// TIA Portal V20 export
// export: Created 2025-12-01T14:56:57.3436706Z, ExportSetting None, DisplayName Totally Integrated Automation Portal, DisplayVersion V20 Update 3, DisplayName TIA Portal Openness, DisplayVersion V20 Update 3, DisplayName TIA Portal Version Control Interface, DisplayVersion V20 Update 3, DisplayName STEP 7 Professional, DisplayVersion V20 Update 3, DisplayName STEP 7 Safety, DisplayVersion V20 Update 2, DisplayName WinCC Basic/Comfort/Advanced, DisplayVersion V20 Update 3, DisplayName WinCC Professional, DisplayVersion V20 Update 3, DisplayName WinCC Unified, DisplayVersion V20 Update 3
FUNCTION_BLOCK "FB376_DesPaletizador_Manual"   // FB376, LAD
TITLE = DesPaletizador Manual (Capas)
{ S7_Optimized_Access := 'FALSE' }
// stored: AutoNumber false, SetENOAutomatically false
   VAR_INPUT
      Maquina : UInt;   // Numero de Maquina
      ConfigDesPaletizador : "UDT_ConfigDesPaletizador";   // DB de Config de Velocidadad
      Robot_Habilitado : Bool;   // ROBOT >> Habilitado
      Robot_OutElevador : Bool;   // ROBOT >> Fuera de la Zona del Elevador
      Robot_PeticionSubir : Bool;   // ROBOT >> Peticion de Subir
      Robot_PeticionBajar : Bool;   // ROBOT >> Peticion de Bajar
      Robot_VelocidadElevador : Int;   // ROBOT >> Velocidad del Elevador
      ByteInicial : Int;   // Byte Inicial del Variador LENZE
      NodoNoPresente : Bool;   // Nodo No Presenye del Variador LENZE
      EnTension : Bool;   // Existe Tension en la Mesa
      Mantenimiento : Bool;   // Llave de Mantenimiento
      TermicoFreno : Bool;   // Termico del Freno
      Seg_UP : Bool;   // Seguridad Abajo de la Elevacion
      Seg_DOWN : Bool;   // Seguridad Abajo de la Elevacion
      pHsPisoCarga : Bool;   // Posicion del Piso de Carga
      pHsPisoDesCarga : Bool;   // Posicion del Piso de DesCarga
      Protrusion : Bool;   // pHs de Protrusion
      P_NuevaCapa : Bool;   // Peticion de Nueva Capa
      P_Subir : Bool;   // Pulsador de Subir
      P_Bajar : Bool;   // Pulsador de Bajar
      BarreraUp : Bool;   // Barrera del Nivel Superior
      pHsAnchura_01 : Bool;
      pHsAnchura_02 : Bool;
      pHsGalibo_01 : Bool;   // pHs de Control de Hueco Superior
      pHsGalibo_02 : Bool;   // pHs de Control de Hueco Superior
      pHsGalibo_03 : Bool;   // pHs de Control de Hueco Superior
      pHsGalibo_04 : Bool;   // pHs de Control de Hueco Superior
      pHsAlturaCota_01 : Bool;
      pHsAlturaCota_02 : Bool;
      pHsAlturaMax_01 : Bool;
      pHsAlturaMax_02 : Bool;
      RoturaCadena_01 : Bool;   // Rotura de Cadena
      RoturaCadena_02 : Bool;   // Rotura de Cadena
      RoturaCadena_03 : Bool;   // Rotura de Cadena
      RoturaCadena_04 : Bool;   // Rotura de Cadena
      FinDesPaletizado : Bool;   // Fin del Paletizado
      SubirManual : Bool;   // Subir en Manual
      BajarManual : Bool;   // Bajar en Manual
      Homming : Bool;
      EncoderIncremental : Bool;
      pHsReferenciaCero : Bool;   // phs de Referencia Cero
      V_TIM_Galibo : Time := T#1S;   // Morgan 14/02/19 500ms ->1s
      V_TIM_Protrusion : Int := 200;
      V_TOut_Elevacion : Int := 15000;
   END_VAR
   VAR_OUTPUT
      DesHabilitarBarreraUp : Bool;   // DesHabilitar Barrerra superior
      H_Puesto : Bool;   // Baliza de Paleta en Puesto
      DI3VarElev_pHsReferenciaCero : Bool;
   END_VAR
   VAR
      PosicionActual : Int;   // Posicion Actual
      PosicionDOWN : Int;   // Interna >> Posicion Abajo
      PosicionUP : Int;   // Interna >> Posicion Arriba
      PosicionOrden : Int;   // Orden >> Posicion A Ejecutar
      PosicionUltima : Int;   // Orden >> Ultima Posicion Enviada
      MemoPosicionActual : Int;   // Memoria >> Altura de la Carga
      MemoEventoDesPaletizado : Int;   // Memoria >> Evento Paletizado
      ConsignaFR : Int;   // Variador >> Consigna
      EstadoElevador : Word;   // Variador >> Estado
      Subject_Area : Word;   // Variador >> Subjet Area
      ID_Area : Word;   // Variador >> ID Area
      Orden : Bool;   // Orden >> Ejecutar
      FinOrden : Bool;   // Orden >> Fin Ejecucion
      PaletaEnPuesto : Bool;   // Interna >> Paleta En el Puesto
      MAQx_SinCapa : Bool;
      MemoCapaDinamico : Bool;
      FP_CapaDinamico : Bool;
      FN_CapaDinamico : Bool;
      InicioCapa : Int;
      FinalCapa : Int;
      MAQx_SinCota : Bool;
      MemoCotaDinamico : Bool;
      FP_CotaDinamico : Bool;
      MA_SubirPuesto : Bool;   // PUESTO >> Subir la Carga
      MA_BajarPuesto : Bool;   // PUESTO >> Bajar la Carga
      MA_Baliza : Bool;   // PUESTO >> Baliza
      PermisoMovElevador : Bool;   // Permiso Mover el Elevador
      PosCarga_OK : Bool;   // Posicionado en Carga
      PosDesCarga_OK : Bool;   // Posicionado en DesCargaCarga
      VarElev_MemoHomingAuto : Bool;   // Variador >>
      VarElev_ReferenciaOK : Bool;   // Variador >>
      VarElev_Error : Bool;   // Variador >>
      EventoInicioDesPaletizado : Bool;   // Evento >> Inicio DesPaletizado
      EventoFinalDesPaletizado : Bool;   // Evento >> Final DesPaletizado
      TIM_EsperaOrden { S7_SetPoint := 'True'} : TON_TIME;   // Orden >> TIM de Espera para Ejecutar
      TMPEnPisoCarga { S7_SetPoint := 'True'} : TON_TIME;
      TMPEnPisoDesCarga { S7_SetPoint := 'True'} : TON_TIME;
      TMP_EnTension { S7_SetPoint := 'True'} : "FB910_CNT_UHS";
      TOut_Elevacion { S7_SetPoint := 'True'} : "FB910_CNT_UHS";
      TIM_Protrusion { S7_SetPoint := 'True'} : "FB910_CNT_UHS";
      TIM_Galibo { S7_SetPoint := 'True'} : TON_TIME;
      TIM_EsperaErrorPosicion { S7_SetPoint := 'True'} : TON_TIME;
   END_VAR
   VAR_TEMP
      EstadoZonaMesa : "EstadoZona";
      EstadoZonaMaquina : "EstadoZona";
      EstadoVI : "EstadosMesa";
      EstadoMAQ : "EstadoMaquina_DesPaletizadoManual";
      DatosScada : "UDT_ScadaDatosMaquina";
      ConfigMAQ : "UDT_ConfigDesPaletizador";
      Auxiliares : Struct
         PosicionAbajo : Int;   // Posicion Abajo del Elevador
         AuxPosMax : Int;
         AuxPosMin : Int;
         Margen : Int;
         AuxAlturaMax : Int;
         AuxAlturaMin : Int;
      END_STRUCT;
      UT_Datos : Struct
         NumeroUT : UInt;
         CotaUT : Int;
         CapaUT : Int;
         SinUT : Bool;
         Con_DestinoUT : Bool;
         OK_DestinoUT : Bool;
      END_STRUCT;
      MovElevador : Struct
         NuevaPosicion : Int;
         AlturaVeloLentisima : Int;
         DestinoDOWN : Bool;   // Moviendose el elevador hacia la posicion de DOWN
         LentaDOWN : Bool;   // Activar velocidad lenta en el moviento hacia la posicion DOWN
         DestinoUP : Bool;   // Moviendose el elevador hacia la posicion de UP
         LentaUP : Bool;   // Activar velocidad lenta en el moviento hacia la posicion UP
         EnPisoAbajo : Bool;
         AlturaMax_OK : Bool;
         AlturaMin_OK : Bool;
      END_STRUCT;
      ZonaEnMarcha : Bool;
      ZonaEnReset : Bool;
      MAQ_Cargada : Bool;
      MAQ_Vacia : Bool;
      AlturaControlBarrerra : Int;
      AlturaCotaDefecto : Int;
      AlturaCapaDefecto : Int;
      AlturaCapaMinima : Int;
      AlturaCapaMaxima : Int;
      TempInt : Int;
   END_VAR
   VAR_TEMP   // added for the SCL form of the ladder/FBD networks
      _w1 : Bool;
      _w2 : Bool;
      _w3 : Bool;
   END_VAR
BEGIN

REGION Network 1: PARAMETROS ESPECIALES
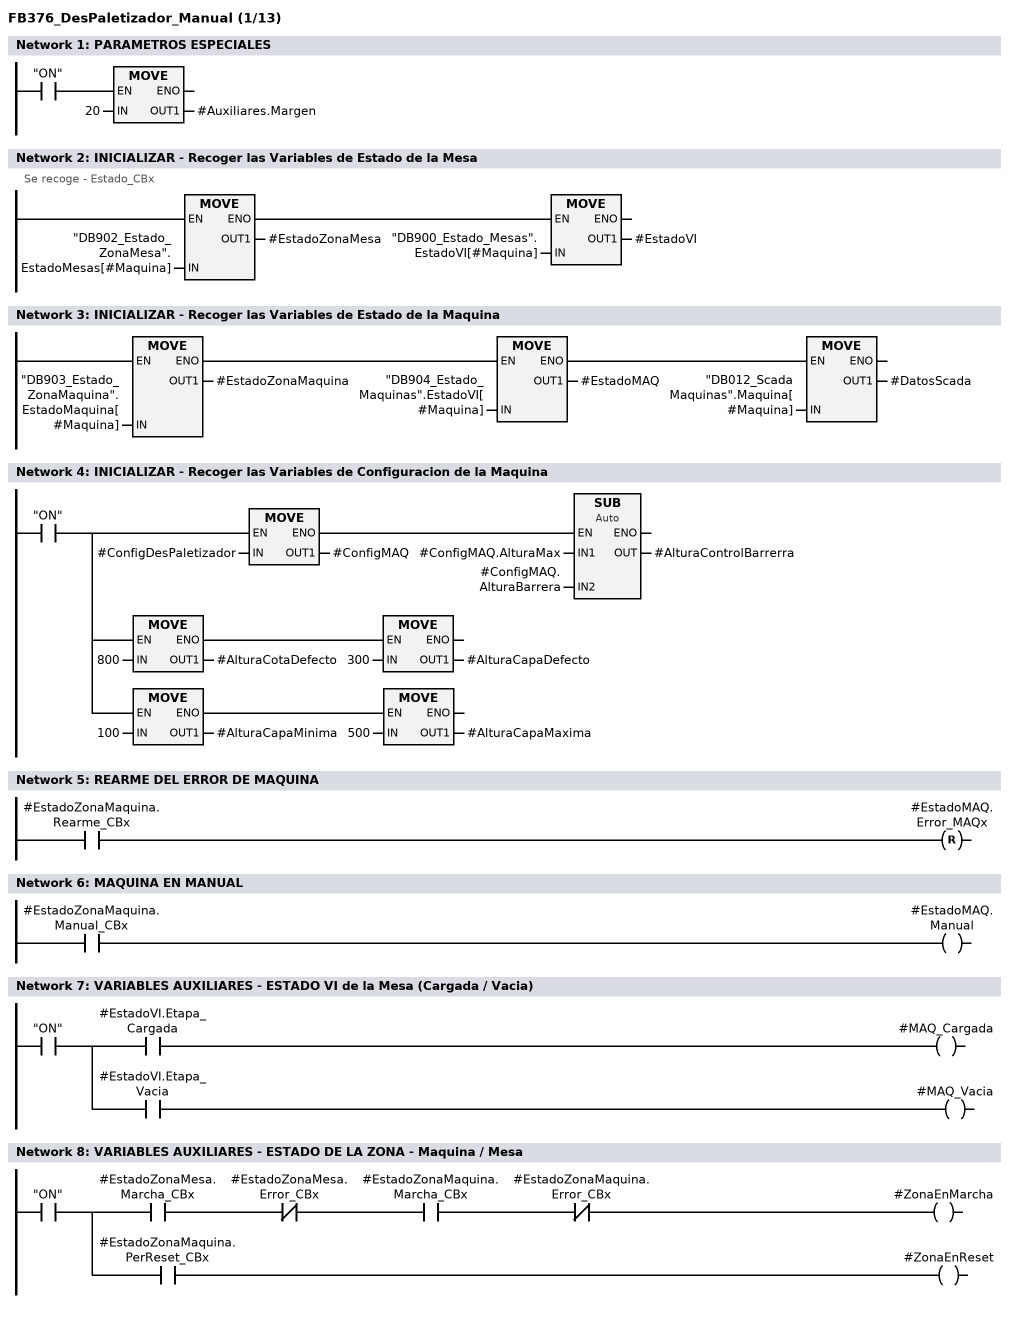
   RUNG wire#powerrail
      Contact( "ON" )
      { S7_GenerateENO := "TRUE" } Move(in := 20, out1 => #Auxiliares.Margen)
   END_RUNG
   // the same network as SCL:
   IF "ON" THEN #Auxiliares.Margen := 20; END_IF;
END_REGION

REGION Network 2: INICIALIZAR - Recoger las Variables de Estado de la Mesa
   // Se recoge - Estado_CBx
   RUNG wire#powerrail
      Move(in := "DB902_Estado_ZonaMesa".EstadoMesas[#Maquina], out1 => #EstadoZonaMesa)
      Move(in := "DB900_Estado_Mesas".EstadoVI[#Maquina], out1 => #EstadoVI)
   END_RUNG
   // the same network as SCL:
   #EstadoZonaMesa := "DB902_Estado_ZonaMesa".EstadoMesas[#Maquina];
   #EstadoVI := "DB900_Estado_Mesas".EstadoVI[#Maquina];
END_REGION

REGION Network 3: INICIALIZAR - Recoger las Variables de Estado de la Maquina
   RUNG wire#powerrail
      Move(in := "DB903_Estado_ZonaMaquina".EstadoMaquina[#Maquina], out1 => #EstadoZonaMaquina)
      Move(in := "DB904_Estado_Maquinas".EstadoVI[#Maquina], out1 => #EstadoMAQ)
      Move(in := "DB012_ScadaMaquinas".Maquina[#Maquina], out1 => #DatosScada)
   END_RUNG
   // the same network as SCL:
   #EstadoZonaMaquina := "DB903_Estado_ZonaMaquina".EstadoMaquina[#Maquina];
   #EstadoMAQ := "DB904_Estado_Maquinas".EstadoVI[#Maquina];
   #DatosScada := "DB012_ScadaMaquinas".Maquina[#Maquina];
END_REGION

REGION Network 4: INICIALIZAR - Recoger las Variables de Configuracion de la Maquina
   RUNG wire#powerrail
      Contact( "ON" )
      wire#w1
      Move(in := #ConfigDesPaletizador, out1 => #ConfigMAQ)
      Sub(in1 := #ConfigMAQ.AlturaMax, in2 := #ConfigMAQ.AlturaBarrera, out => #AlturaControlBarrerra)
   END_RUNG
   RUNG wire#w1
      Move(in := 800, out1 => #AlturaCotaDefecto)
      Move(in := 300, out1 => #AlturaCapaDefecto)
   END_RUNG
   RUNG wire#w1
      Move(in := 100, out1 => #AlturaCapaMinima)
      Move(in := 500, out1 => #AlturaCapaMaxima)
   END_RUNG
   // the same network as SCL:
   IF "ON" THEN
       #ConfigMAQ := #ConfigDesPaletizador;
       #AlturaControlBarrerra := #ConfigMAQ.AlturaMax - #ConfigMAQ.AlturaBarrera;
       #AlturaCotaDefecto := 800;
       #AlturaCapaDefecto := 300;
       #AlturaCapaMinima := 100;
       #AlturaCapaMaxima := 500;
   END_IF;
END_REGION

REGION Network 5: REARME DEL ERROR DE MAQUINA
   RUNG wire#powerrail
      Contact( #EstadoZonaMaquina.Rearme_CBx )
      R_Coil( #EstadoMAQ.Error_MAQx )
   END_RUNG
   // the same network as SCL:
   IF #EstadoZonaMaquina.Rearme_CBx THEN #EstadoMAQ.Error_MAQx := FALSE; END_IF;
END_REGION

REGION Network 6: MAQUINA EN MANUAL
   RUNG wire#powerrail
      Contact( #EstadoZonaMaquina.Manual_CBx )
      Coil( #EstadoMAQ.Manual )
   END_RUNG
   // the same network as SCL:
   #EstadoMAQ.Manual := #EstadoZonaMaquina.Manual_CBx;
END_REGION

REGION Network 7: VARIABLES AUXILIARES - ESTADO VI de la Mesa (Cargada / Vacia)
   RUNG wire#powerrail
      Contact( "ON" )
      wire#w1
      Contact( #EstadoVI.Etapa_Cargada )
      Coil( #MAQ_Cargada )
   END_RUNG
   RUNG wire#w1
      Contact( #EstadoVI.Etapa_Vacia )
      Coil( #MAQ_Vacia )
   END_RUNG
   // the same network as SCL:
   #MAQ_Cargada := "ON" AND #EstadoVI.Etapa_Cargada;
   #MAQ_Vacia := "ON" AND #EstadoVI.Etapa_Vacia;
END_REGION

REGION Network 8: VARIABLES AUXILIARES - ESTADO DE LA ZONA - Maquina / Mesa
   RUNG wire#powerrail
      Contact( "ON" )
      wire#w1
      Contact( #EstadoZonaMesa.Marcha_CBx )
      I_Contact( #EstadoZonaMesa.Error_CBx )
      Contact( #EstadoZonaMaquina.Marcha_CBx )
      I_Contact( #EstadoZonaMaquina.Error_CBx )
      Coil( #ZonaEnMarcha )
   END_RUNG
   RUNG wire#w1
      Contact( #EstadoZonaMaquina.PerReset_CBx )
      Coil( #ZonaEnReset )
   END_RUNG
   // the same network as SCL:
   #ZonaEnMarcha := "ON" AND #EstadoZonaMesa.Marcha_CBx AND NOT #EstadoZonaMesa.Error_CBx AND #EstadoZonaMaquina.Marcha_CBx AND NOT #EstadoZonaMaquina.Error_CBx;
   #ZonaEnReset := "ON" AND #EstadoZonaMaquina.PerReset_CBx;
END_REGION

NETWORK
TITLE = CONTROL DE RESET de Variables Auxiliares
/////////////////////////////////////////////////////////////////////////////
/////////////////////////////////////////////////////////////////////////////
// --- Si realiza un RESET hay que limpiar las variables

      SET;  // Reseteando la Maquina ?
      AN    #ZonaEnReset;
      JC    NoExiste_Reset;

      SET;
      R     #Orden;
      R     #PaletaEnPuesto;  // Variable del Puesto de Trabajo
      R     #MAQx_SinCota;
      R     #MAQx_SinCapa;

      L     0;
      T     #PosicionOrden;

NoExiste_Reset:NOP   0;



NETWORK
TITLE = CONTROL DE MOVIMIENTO DEL ELEVADOR - PROTOCOLO
/////////////////////////////////////////////////////////////////////////////
/////////////////////////////////////////////////////////////////////////////
// ---  Cierre del Protocolo

      SET;
      O     #Orden;  // - Hay que protocolo la Orden
      O     #FinOrden;  //   en ejecucion
      JCN   Final_ProtocoloOrden;
      SET;
      A     #Orden;  // - Hay que protocolo la Orden
      A     #FinOrden;  //   en ejecucion
      JCN   Final_ProtocoloOrden;

      L     0;  // -- Resetear Variables
      T     #PosicionOrden;

      SET;
      R     #Orden;

      JU    Final_ProtocoloOrden;


/////////////////////////////////////////////////////////////////////////////
/////////////////////////////////////////////////////////////////////////////
// ---  Final del Control

Final_ProtocoloOrden:NOP   0;


NETWORK
TITLE = RECOGER DATOS EXISTENTES DE LA UT
/////////////////////////////////////////////////////////////////////////////
/////////////////////////////////////////////////////////////////////////////
// ---  Datos de la UT en la Maquina
      L     0;
      T     #UT_Datos.CotaUT;
      T     #UT_Datos.CapaUT;

      SET;  // - Incializar datos de la UT
      R     #UT_Datos.OK_DestinoUT;
      R     #UT_Datos.Con_DestinoUT;
      S     #UT_Datos.SinUT;


/////////////////////////////////////////////////////////////////////////////
/////////////////////////////////////////////////////////////////////////////
// --- Comprobar si existen UT en la Mesa = Maquina

      L     "DB810_ColasMesas".Colas[#Maquina].UT_PrimeraMesa;
      T     #UT_Datos.NumeroUT;

      SET;  // No hay UT's ?
      L     #UT_Datos.NumeroUT;
      L     0;
      ==I;
      JC    Final_DatosUT;


/////////////////////////////////////////////////////////////////////////////
/////////////////////////////////////////////////////////////////////////////
// --- Recoger Datos
      SET;
      R     #UT_Datos.SinUT;  // --- Hay UT

      L     "DB815_UTs_Datos".UT[#UT_Datos.NumeroUT].CotaAltura;
      T     #UT_Datos.CotaUT;  // Altura de la Carga
      L     "DB815_UTs_Datos".UT[#UT_Datos.NumeroUT].Amarre;
      T     #UT_Datos.CapaUT;  // Capa

      SET;  // --- Comprobacion de Destino
      L     "DB812_UTs_Control".UT[#UT_Datos.NumeroUT].MesaDestino;
      L     0;
      ==I;
      JC    NoExiste_Destino;

      SET;  // --- Tiene Destino
      S     #UT_Datos.Con_DestinoUT;

      SET;  // --- Existe Destino de Evacuacion
      L     "DB812_UTs_Control".UT[#UT_Datos.NumeroUT].MesaDestino;
      L     "DB812_UTs_Control".UT[#UT_Datos.NumeroUT].MesaActual;
      <>I;
      S     #UT_Datos.OK_DestinoUT;

NoExiste_Destino:NOP   0;



/////////////////////////////////////////////////////////////////////////////
/////////////////////////////////////////////////////////////////////////////
// --- Control de la Altura de la UT

      L     #UT_Datos.CotaUT;  // - Control de la Cota
      L     0;
      <>I;
      JC    Existe_CotaUT;

      SET;
      S     #MAQx_SinCota;  // - Cota dianamica

      L     #AlturaCotaDefecto;  // - Valor de Defecto
      T     #UT_Datos.CotaUT;  // Se guarda ?
//      T     "DB815_DatosUT".Datos_UTs[#NumeroUT].CotaAltura

Existe_CotaUT:NOP   0;


/////////////////////////////////////////////////////////////////////////////
/////////////////////////////////////////////////////////////////////////////
// --- Control de la Capa de la UT

      L     #UT_Datos.CapaUT;  // - Control de la Capa
      L     0;
      <>I;
      JC    Existe_CapaUT;

      SET;
      S     #MAQx_SinCapa;  // - Capa dianamica

      L     #AlturaCapaDefecto;  //   Valor de Defecto
      T     #UT_Datos.CapaUT;  // Se guarda ?
      T     "DB815_UTs_Datos".UT[#UT_Datos.NumeroUT].Amarre;


Existe_CapaUT:NOP   0;
// - Altura para DesActivar el control de la Barrera
      L     #UT_Datos.CapaUT;
      L     200;
      +I;
      T     #AlturaControlBarrerra;


/////////////////////////////////////////////////////////////////////////////
/////////////////////////////////////////////////////////////////////////////
// --- Datos Recogidos
Final_DatosUT:NOP   0;  // --- Fin de los Datos de la UT

      SET;  // --- Configuracion del DesPaletizador
      AN    #UT_Datos.SinUT;  //     Dinamico
      JC    Existe_UT;

      R     #MAQx_SinCota;
      R     #MAQx_SinCapa;

Existe_UT:NOP   0;



REGION Network 12: VARIABLES AUXILIARES - Calculo de la Posicion Abajo del Elevador
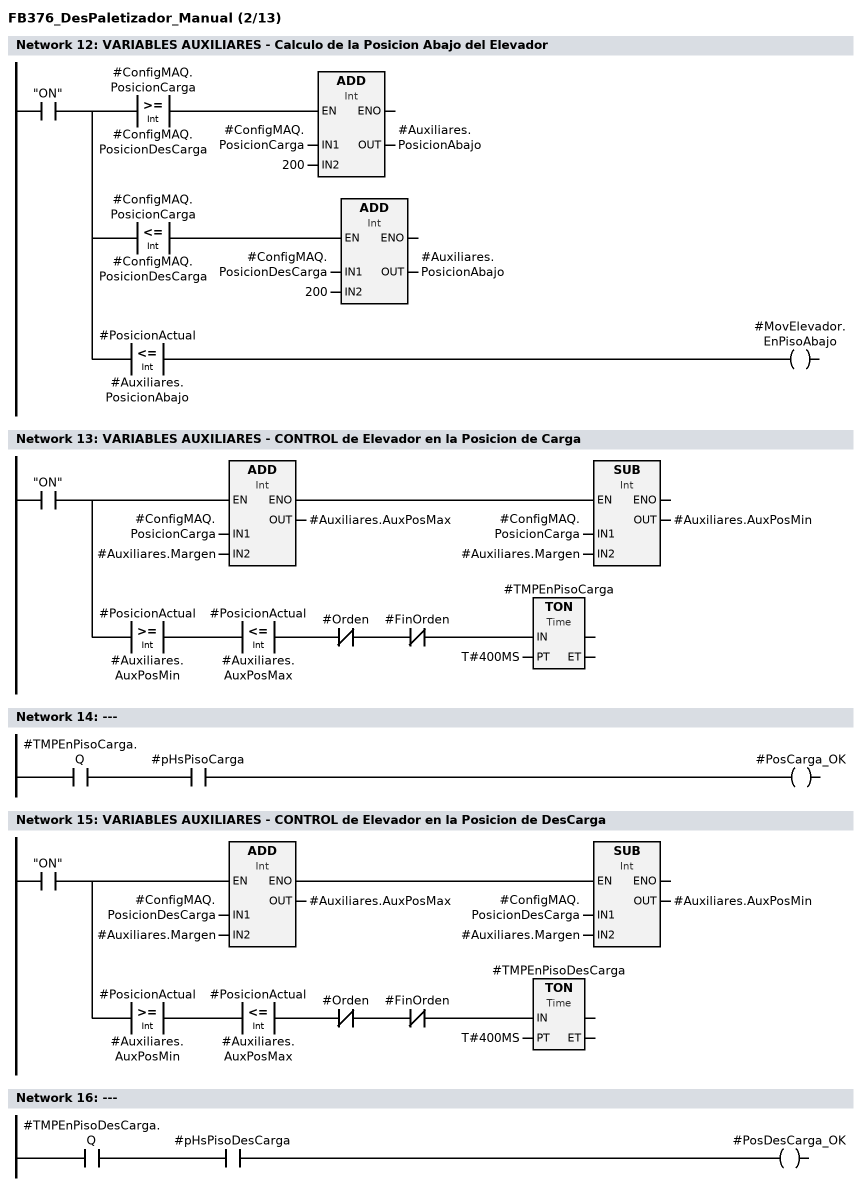
   RUNG wire#powerrail
      Contact( "ON" )
      wire#w1
      { S7_Templates := "SrcType := Int" } GE_Contact(in1 := #ConfigMAQ.PosicionCarga, in2 := #ConfigMAQ.PosicionDesCarga)
      { S7_Templates := "SrcType := Int"; S7_GenerateENO := "TRUE" } Add(in1 := #ConfigMAQ.PosicionCarga, in2 := 200, out => #Auxiliares.PosicionAbajo)
   END_RUNG
   RUNG wire#w1
      { S7_Templates := "SrcType := Int" } LE_Contact(in1 := #ConfigMAQ.PosicionCarga, in2 := #ConfigMAQ.PosicionDesCarga)
      { S7_Templates := "SrcType := Int"; S7_GenerateENO := "TRUE" } Add(in1 := #ConfigMAQ.PosicionDesCarga, in2 := 200, out => #Auxiliares.PosicionAbajo)
   END_RUNG
   RUNG wire#w1
      { S7_Templates := "SrcType := Int" } LE_Contact(in1 := #PosicionActual, in2 := #Auxiliares.PosicionAbajo)
      Coil( #MovElevador.EnPisoAbajo )
   END_RUNG
   // the same network as SCL:
   IF "ON" AND (#ConfigMAQ.PosicionCarga >= #ConfigMAQ.PosicionDesCarga) THEN
       #Auxiliares.PosicionAbajo := #ConfigMAQ.PosicionCarga + 200;
   END_IF;
   IF "ON" AND (#ConfigMAQ.PosicionCarga <= #ConfigMAQ.PosicionDesCarga) THEN
       #Auxiliares.PosicionAbajo := #ConfigMAQ.PosicionDesCarga + 200;
   END_IF;
   #MovElevador.EnPisoAbajo := "ON" AND (#PosicionActual <= #Auxiliares.PosicionAbajo);
END_REGION

REGION Network 13: VARIABLES AUXILIARES - CONTROL de Elevador en la Posicion de Carga
   RUNG wire#powerrail
      Contact( "ON" )
      wire#w1
      { S7_Templates := "SrcType := Int"; S7_GenerateENO := "TRUE" } Add(in1 := #ConfigMAQ.PosicionCarga, in2 := #Auxiliares.Margen, out => #Auxiliares.AuxPosMax)
      { S7_Templates := "SrcType := Int"; S7_GenerateENO := "TRUE" } Sub(in1 := #ConfigMAQ.PosicionCarga, in2 := #Auxiliares.Margen, out => #Auxiliares.AuxPosMin)
   END_RUNG
   RUNG wire#w1
      { S7_Templates := "SrcType := Int" } GE_Contact(in1 := #PosicionActual, in2 := #Auxiliares.AuxPosMin)
      { S7_Templates := "SrcType := Int" } LE_Contact(in1 := #PosicionActual, in2 := #Auxiliares.AuxPosMax)
      I_Contact( #Orden )
      I_Contact( #FinOrden )
      { S7_Templates := "time_type := Time" } #TMPEnPisoCarga.TON(pt := T#400MS, et =>)
   END_RUNG
   // the same network as SCL:
   // ENO of a box is taken as its EN; it also drops when the box reports an error
   IF "ON" THEN
       #Auxiliares.AuxPosMax := #ConfigMAQ.PosicionCarga + #Auxiliares.Margen;
       #Auxiliares.AuxPosMin := #ConfigMAQ.PosicionCarga - #Auxiliares.Margen;
   END_IF;
   #TMPEnPisoCarga(IN := "ON" AND (#PosicionActual >= #Auxiliares.AuxPosMin) AND (#PosicionActual <= #Auxiliares.AuxPosMax) AND NOT #Orden AND NOT #FinOrden,   // TON
                   PT := T#400MS);
END_REGION

REGION Network 14: ---
   RUNG wire#powerrail
      Contact( #TMPEnPisoCarga.Q )
      Contact( #pHsPisoCarga )
      Coil( #PosCarga_OK )
   END_RUNG
   // the same network as SCL:
   #PosCarga_OK := #TMPEnPisoCarga.Q AND #pHsPisoCarga;
END_REGION

REGION Network 15: VARIABLES AUXILIARES - CONTROL de Elevador en la Posicion de DesCarga
   RUNG wire#powerrail
      Contact( "ON" )
      wire#w1
      { S7_Templates := "SrcType := Int"; S7_GenerateENO := "TRUE" } Add(in1 := #ConfigMAQ.PosicionDesCarga, in2 := #Auxiliares.Margen, out => #Auxiliares.AuxPosMax)
      { S7_Templates := "SrcType := Int"; S7_GenerateENO := "TRUE" } Sub(in1 := #ConfigMAQ.PosicionDesCarga, in2 := #Auxiliares.Margen, out => #Auxiliares.AuxPosMin)
   END_RUNG
   RUNG wire#w1
      { S7_Templates := "SrcType := Int" } GE_Contact(in1 := #PosicionActual, in2 := #Auxiliares.AuxPosMin)
      { S7_Templates := "SrcType := Int" } LE_Contact(in1 := #PosicionActual, in2 := #Auxiliares.AuxPosMax)
      I_Contact( #Orden )
      I_Contact( #FinOrden )
      { S7_Templates := "time_type := Time" } #TMPEnPisoDesCarga.TON(pt := T#400MS, et =>)
   END_RUNG
   // the same network as SCL:
   // ENO of a box is taken as its EN; it also drops when the box reports an error
   IF "ON" THEN
       #Auxiliares.AuxPosMax := #ConfigMAQ.PosicionDesCarga + #Auxiliares.Margen;
       #Auxiliares.AuxPosMin := #ConfigMAQ.PosicionDesCarga - #Auxiliares.Margen;
   END_IF;
   #TMPEnPisoDesCarga(IN := "ON" AND (#PosicionActual >= #Auxiliares.AuxPosMin) AND (#PosicionActual <= #Auxiliares.AuxPosMax) AND NOT #Orden AND NOT #FinOrden,   // TON
                      PT := T#400MS);
END_REGION

REGION Network 16: ---
   RUNG wire#powerrail
      Contact( #TMPEnPisoDesCarga.Q )
      Contact( #pHsPisoDesCarga )
      Coil( #PosDesCarga_OK )
   END_RUNG
   // the same network as SCL:
   #PosDesCarga_OK := #TMPEnPisoDesCarga.Q AND #pHsPisoDesCarga;
END_REGION

REGION Network 17: VARIABLES AUXILIARES - CONTROL de Movimiento del Elevador en el Puesto de Trabajo (Maximo y Minimo)
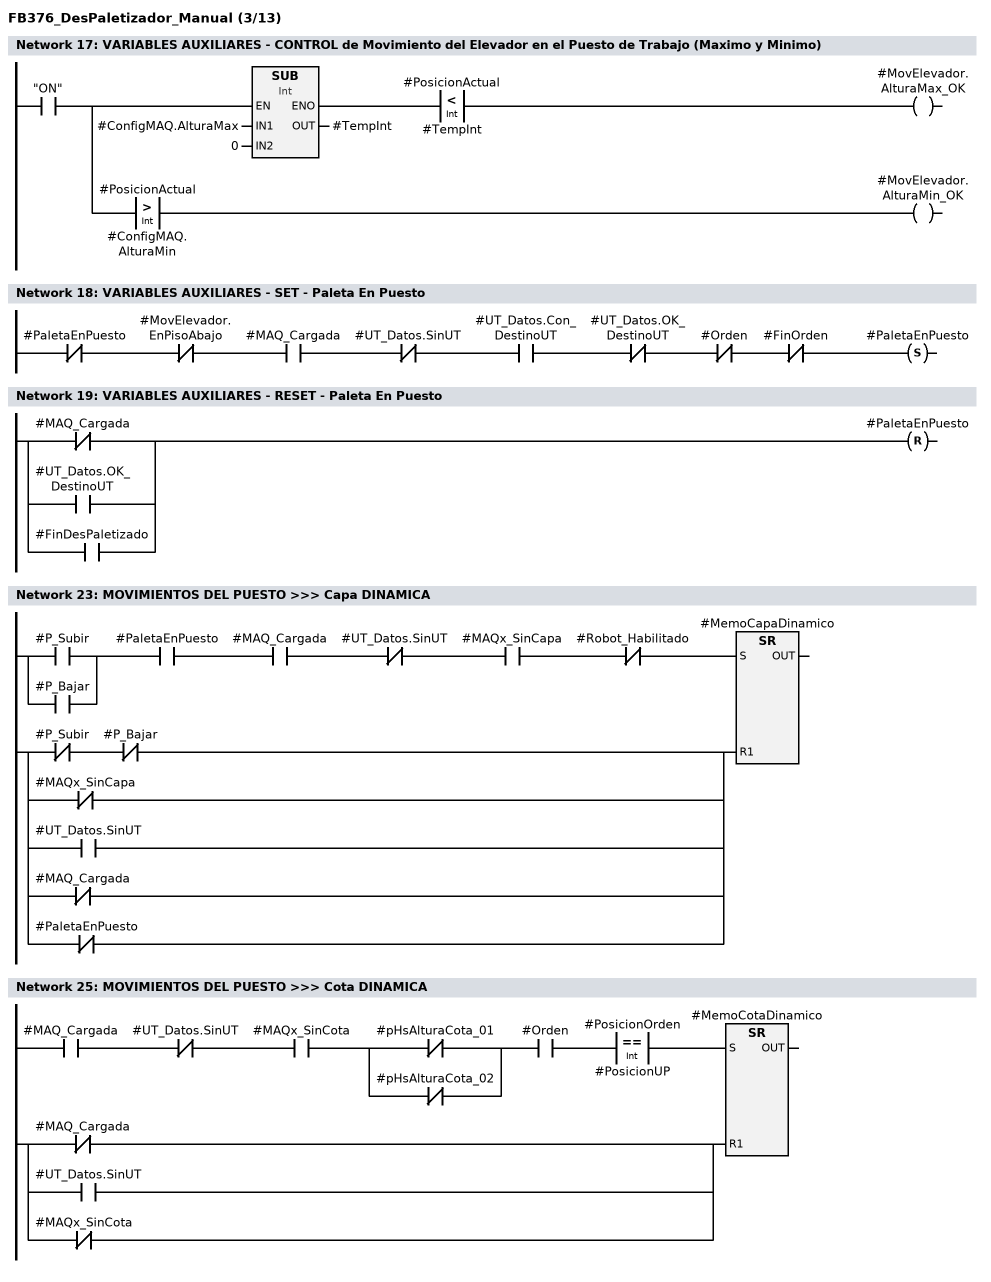
   RUNG wire#powerrail
      Contact( "ON" )
      wire#w1
      { S7_Templates := "SrcType := Int"; S7_GenerateENO := "TRUE" } Sub(in1 := #ConfigMAQ.AlturaMax, in2 := 0, out => #TempInt)
      { S7_Templates := "SrcType := Int" } LT_Contact(in1 := #PosicionActual, in2 := #TempInt)
      Coil( #MovElevador.AlturaMax_OK )
   END_RUNG
   RUNG wire#w1
      { S7_Templates := "SrcType := Int" } GT_Contact(in1 := #PosicionActual, in2 := #ConfigMAQ.AlturaMin)
      Coil( #MovElevador.AlturaMin_OK )
   END_RUNG
   // the same network as SCL:
   // ENO of a box is taken as its EN; it also drops when the box reports an error
   IF "ON" THEN #TempInt := #ConfigMAQ.AlturaMax - 0; END_IF;
   #MovElevador.AlturaMax_OK := "ON" AND (#PosicionActual < #TempInt);
   #MovElevador.AlturaMin_OK := "ON" AND (#PosicionActual > #ConfigMAQ.AlturaMin);
END_REGION

REGION Network 18: VARIABLES AUXILIARES - SET - Paleta En Puesto
   RUNG wire#powerrail
      I_Contact( #PaletaEnPuesto )
      I_Contact( #MovElevador.EnPisoAbajo )
      Contact( #MAQ_Cargada )
      I_Contact( #UT_Datos.SinUT )
      Contact( #UT_Datos.Con_DestinoUT )
      I_Contact( #UT_Datos.OK_DestinoUT )
      I_Contact( #Orden )
      I_Contact( #FinOrden )
      S_Coil( #PaletaEnPuesto )
   END_RUNG
   // the same network as SCL:
   IF NOT #PaletaEnPuesto AND NOT #MovElevador.EnPisoAbajo AND #MAQ_Cargada AND NOT #UT_Datos.SinUT AND #UT_Datos.Con_DestinoUT AND NOT #UT_Datos.OK_DestinoUT AND NOT #Orden AND NOT #FinOrden THEN
       #PaletaEnPuesto := TRUE;
   END_IF;
END_REGION

REGION Network 19: VARIABLES AUXILIARES - RESET - Paleta En Puesto
   RUNG wire#powerrail
      I_Contact( #MAQ_Cargada )
      wire#w1
      R_Coil( #PaletaEnPuesto )
   END_RUNG
   RUNG wire#powerrail
      Contact( #UT_Datos.OK_DestinoUT )
   END_RUNG wire#w1
   RUNG wire#powerrail
      Contact( #FinDesPaletizado )
   END_RUNG wire#w1
   // the same network as SCL:
   IF NOT #MAQ_Cargada OR #UT_Datos.OK_DestinoUT OR #FinDesPaletizado THEN #PaletaEnPuesto := FALSE; END_IF;
END_REGION

NETWORK
TITLE = MOVIMIENTOS DEL PUESTO >>> Control de Nueva CAPA
/////////////////////////////////////////////////////////////////////////////
/////////////////////////////////////////////////////////////////////////////
// ---  CONTROL DE NUEVA CAPA
      SET;
      A     #P_NuevaCapa;  // --- Se pulsado Nueva Capa ?
      A     #PaletaEnPuesto;  //     cuando esta la Paleta en el Puesto
      A     #MAQ_Cargada;  // --- Controles
      AN    #UT_Datos.SinUT;
      AN    #UT_Datos.OK_DestinoUT;
      AN    #FinDesPaletizado;
      AN    #Orden;
      AN    #FinOrden;
      AN    #Robot_Habilitado;
      JCN   Fin_ControlNuevaCapa;  // --- Realizar Nueva Capa ?


/////////////////////////////////////////////////////////////////////////////
/////////////////////////////////////////////////////////////////////////////
/////////////////////////////////////////////////////////////////////////////
      L     #PosicionActual;  // --- Calcular nueva posicion de parada
      L     #UT_Datos.CapaUT;  //     + Altura de Capa
      +D;
      T     #MovElevador.NuevaPosicion;

      L     #MovElevador.NuevaPosicion;  // --- Comprueba que no sobrepasa la altura maxima
      L     #ConfigMAQ.AlturaMax;
      <=I;
      JC    EjecutarOrden_NuevaCapa;

      L     #ConfigMAQ.AlturaMax;  // Lo maximo que se posiciona
      T     #MovElevador.NuevaPosicion;  // para trabajar

EjecutarOrden_NuevaCapa:NOP   0;
      L     #MovElevador.NuevaPosicion;
      T     #PosicionUP;  // - Guardar la Posicion UP
      T     #PosicionOrden;
      T     #PosicionUltima;

      S     #Orden;


/////////////////////////////////////////////////////////////////////////////
/////////////////////////////////////////////////////////////////////////////
/////////////////////////////////////////////////////////////////////////////
Fin_ControlNuevaCapa:NOP   0;



NETWORK
TITLE = CONTROL DE PULSADOR DE Subir >>> MA_SubirPuesto
/////////////////////////////////////////////////////////////////////////////
/////////////////////////////////////////////////////////////////////////////
// ---  Movimientos manuales desde el Puesto >>> SUBIR
      SET;
      A     #P_Subir;  // --- Orden de Subir el Elevador
      AN    #P_Bajar;
      AN    #P_NuevaCapa;
      A     #MovElevador.AlturaMax_OK;
      A     #PaletaEnPuesto;
      A     #MAQ_Cargada;  // --- Controles
      AN    #UT_Datos.SinUT;
      AN    #UT_Datos.OK_DestinoUT;
      AN    #FinDesPaletizado;
      AN    #Orden;
      AN    #FinOrden;
      AN    #Robot_Habilitado;
      =     #MA_SubirPuesto;




NETWORK
TITLE = CONTROL DE PULSADOR DE Bajar >>> MA_BajarPuesto
/////////////////////////////////////////////////////////////////////////////
/////////////////////////////////////////////////////////////////////////////
// ---  Movimientos manuales desde el Puesto >>> BAJAR
      SET;
      AN    #P_Subir;  // --- Orden de Bajar el Elevador
      A     #P_Bajar;
      AN    #P_NuevaCapa;
      A     #MovElevador.AlturaMin_OK;
      A     #PaletaEnPuesto;
      A     #MAQ_Cargada;  // --- Controles
      AN    #UT_Datos.SinUT;
      AN    #UT_Datos.OK_DestinoUT;
      AN    #FinDesPaletizado;
      AN    #Orden;
      AN    #FinOrden;
      AN    #Robot_Habilitado;
      =     #MA_BajarPuesto;



REGION Network 23: MOVIMIENTOS DEL PUESTO >>> Capa DINAMICA
   RUNG wire#powerrail
      Contact( #P_Subir )
      wire#w1
      Contact( #PaletaEnPuesto )
      Contact( #MAQ_Cargada )
      I_Contact( #UT_Datos.SinUT )
      Contact( #MAQx_SinCapa )
      I_Contact( #Robot_Habilitado )
      S_SR(operand := #MemoCapaDinamico, r1 := wire#w2)
   END_RUNG
   RUNG wire#powerrail
      Contact( #P_Bajar )
   END_RUNG wire#w1
   RUNG wire#powerrail
      I_Contact( #P_Subir )
      I_Contact( #P_Bajar )
   END_RUNG wire#w2
   RUNG wire#powerrail
      I_Contact( #MAQx_SinCapa )
   END_RUNG wire#w2
   RUNG wire#powerrail
      Contact( #UT_Datos.SinUT )
   END_RUNG wire#w2
   RUNG wire#powerrail
      I_Contact( #MAQ_Cargada )
   END_RUNG wire#w2
   RUNG wire#powerrail
      I_Contact( #PaletaEnPuesto )
   END_RUNG wire#w2
   // the same network as SCL:
   IF (#P_Subir OR #P_Bajar) AND #PaletaEnPuesto AND #MAQ_Cargada AND NOT #UT_Datos.SinUT AND #MAQx_SinCapa AND NOT #Robot_Habilitado THEN
       #MemoCapaDinamico := TRUE;   // SR flip-flop
   END_IF;
   IF (NOT #P_Subir AND NOT #P_Bajar) OR NOT #MAQx_SinCapa OR #UT_Datos.SinUT OR NOT #MAQ_Cargada OR NOT #PaletaEnPuesto THEN
       #MemoCapaDinamico := FALSE;
   END_IF;
END_REGION

NETWORK
TITLE = ---
/////////////////////////////////////////////////////////////////////////////
/////////////////////////////////////////////////////////////////////////////
/////////////////////////////////////////////////////////////////////////////
// --- Control Iniciales
      SET;  // --- Mirar Si existe control dianimico de CAPA
      AN    #MAQx_SinCapa;
      JC    Final_ControlCapaDinamica;
      SET;  // --- Existe UT
      A     #UT_Datos.SinUT;
      JC    Final_ControlCapaDinamica;


/////////////////////////////////////////////////////////////////////////////
/////////////////////////////////////////////////////////////////////////////
/////////////////////////////////////////////////////////////////////////////
// --- Control del Calculo de Capa Dinamica
      SET;
      A     #MemoCapaDinamico;
      FP    #FP_CapaDinamico;  // --- FP del Calculo de Capa
      JC    Inicio_CalculoCapaDianamica;

      SET;
      A     #MemoCapaDinamico;
      FN    #FN_CapaDinamico;  // --- FP del Calculo de Capa
      JC    Final_CalculoCapaDianamica;

      JU    Final_ControlCapaDinamica;


/////////////////////////////////////////////////////////////////////////////
/////////////////////////////////////////////////////////////////////////////
/////////////////////////////////////////////////////////////////////////////
//--- Inicio del Calculo de Capa
Inicio_CalculoCapaDianamica:NOP   0;
      L     #PosicionActual;
      T     #InicioCapa;
      JU    Final_ControlCapaDinamica;


/////////////////////////////////////////////////////////////////////////////
/////////////////////////////////////////////////////////////////////////////
/////////////////////////////////////////////////////////////////////////////
//--- Fin del Calculo de Capa
Final_CalculoCapaDianamica:NOP   0;
      L     #PosicionActual;
      T     #FinalCapa;

      L     #FinalCapa;  // --- Altura de nueva capa
      L     #InicioCapa;
      -I;
      L     #UT_Datos.CapaUT;
      +I;
      T     #UT_Datos.CapaUT;

/////////////////////////////////////////////////////////////////////////////
//--- Altura Minima de Capa ? (Altura Capa Minima)
      L     #UT_Datos.CapaUT;
      L     #AlturaCapaMinima;
      >=I;
      JC    MimimoOK_ControlCapaDinamica;

      L     #AlturaCapaMinima;
      T     #UT_Datos.CapaUT;
MimimoOK_ControlCapaDinamica:NOP   0;

/////////////////////////////////////////////////////////////////////////////
//--- Altura Maxima de Capa ? (Altura Capa Maxima)
      L     #UT_Datos.CapaUT;  // --- Altura MAxima de Capa
      L     #AlturaCapaMaxima;  //     Max.Capa por defecto
      <=I;
      JC    MaximoOK_ControlCapaDinamica;

      L     #AlturaCapaMaxima;
      T     #UT_Datos.CapaUT;
MaximoOK_ControlCapaDinamica:NOP   0;

//--- Guardar la Nueva Capa de la UT
      L     #UT_Datos.CapaUT;
      T     "DB815_UTs_Datos".UT[#UT_Datos.NumeroUT].Amarre;


/////////////////////////////////////////////////////////////////////////////
/////////////////////////////////////////////////////////////////////////////
/////////////////////////////////////////////////////////////////////////////
Final_ControlCapaDinamica:NOP   0;



REGION Network 25: MOVIMIENTOS DEL PUESTO >>> Cota DINAMICA
   RUNG wire#powerrail
      Contact( #MAQ_Cargada )
      I_Contact( #UT_Datos.SinUT )
      Contact( #MAQx_SinCota )
      wire#w1
      I_Contact( #pHsAlturaCota_01 )
      wire#w2
      Contact( #Orden )
      { S7_Templates := "SrcType := Int" } EQ_Contact(in1 := #PosicionOrden, in2 := #PosicionUP)
      S_SR(operand := #MemoCotaDinamico, r1 := wire#w3)
   END_RUNG
   RUNG wire#w1
      I_Contact( #pHsAlturaCota_02 )
   END_RUNG wire#w2
   RUNG wire#powerrail
      I_Contact( #MAQ_Cargada )
   END_RUNG wire#w3
   RUNG wire#powerrail
      Contact( #UT_Datos.SinUT )
   END_RUNG wire#w3
   RUNG wire#powerrail
      I_Contact( #MAQx_SinCota )
   END_RUNG wire#w3
   // the same network as SCL:
   IF #MAQ_Cargada AND NOT #UT_Datos.SinUT AND #MAQx_SinCota AND (NOT #pHsAlturaCota_01 OR NOT #pHsAlturaCota_02) AND #Orden AND (#PosicionOrden = #PosicionUP) THEN
       #MemoCotaDinamico := TRUE;   // SR flip-flop
   END_IF;
   IF NOT #MAQ_Cargada OR #UT_Datos.SinUT OR NOT #MAQx_SinCota THEN #MemoCotaDinamico := FALSE; END_IF;
END_REGION

NETWORK
TITLE = ---
/////////////////////////////////////////////////////////////////////////////
/////////////////////////////////////////////////////////////////////////////
/////////////////////////////////////////////////////////////////////////////
// --- Control Iniciales
      SET;  // --- Mirar Si existe control dianimico de Cota
      AN    #MAQx_SinCota;
      JC    Final_ControlCotaDinamica;
      SET;  // --- Existe UT
      A     #UT_Datos.SinUT;
      JC    Final_ControlCotaDinamica;


/////////////////////////////////////////////////////////////////////////////
/////////////////////////////////////////////////////////////////////////////
/////////////////////////////////////////////////////////////////////////////
// --- Control de Altura de la Paleta COTA--> Solo la primera vez
      SET;
      A     #MemoCotaDinamico;
      FP    #FP_CotaDinamico;  // --- FP del Calculo de Cota
      JCN   Final_ControlCotaDinamica;

/////////////////////////////////////////////////////////////////////////////
// --- Nueva Posicion de Parada
      L     #ConfigMAQ.AlturaMax;
      L     #ConfigMAQ.AlturaGalibo;
      -I;
      L     #PosicionActual;
      +I;
      L     #UT_Datos.CapaUT;
      +I;
//     L     #AlturaPaleta        // --- NO NECESARIO ???
//      +I
      T     #MovElevador.NuevaPosicion;

/////////////////////////////////////////////////////////////////////////////
//--- Altura Maxima de Cota ? (Altura Maxima)
      L     #MovElevador.NuevaPosicion;  // --- Comprueba que no sobrepasa
      L     #ConfigMAQ.AlturaMax;  //     la altura maxima
      <=I;
      JC    MaximoOK_ControlCotaDinamica;

      L     #ConfigMAQ.AlturaMax;  // Lo maximo que se posiciona
      T     #MovElevador.NuevaPosicion;  // para trabajar

MaximoOK_ControlCotaDinamica:NOP   0;
      L     #MovElevador.NuevaPosicion;
      T     #PosicionOrden;
      T     #PosicionUltima;
      T     #PosicionUP;


/////////////////////////////////////////////////////////////////////////////
/////////////////////////////////////////////////////////////////////////////
/////////////////////////////////////////////////////////////////////////////
Final_ControlCotaDinamica:NOP   0;



NETWORK
TITLE = GESTION DE ORDENES DE POSICIONADO >>> POSICIONAR el Elevador --- Controles Iniciales
/////////////////////////////////////////////////////////////////////////////
/////////////////////////////////////////////////////////////////////////////
// --- Controles iniciales
      SET;  // Ya esta la Paleta en el Puesto ?
      A     #PaletaEnPuesto;
      JC    Final_ControlOrdenes;

      SET;  // Esta en Marcha ?
      AN    #ZonaEnMarcha;
      JC    Final_ControlOrdenes;

      SET;  // Hay Orden en Curso ?
      A     #Orden;
      O     #FinOrden;
      JC    Final_ControlOrdenes;




NETWORK
TITLE = ---- Distribucion para Ordenes de Posicionado
/////////////////////////////////////////////////////////////////////////////
/////////////////////////////////////////////////////////////////////////////
/////////////////////////////////////////////////////////////////////////////
/////////////////////////////////////////////////////////////////////////////
// --- CONTROL DE ORDENES >>> La Paleta No esta en el Puesto


// --- Posicionar para CARGAR
      SET;
      A     #MAQ_Vacia;  // Esta VACIA
      A     #UT_Datos.SinUT;  // No hay UT
      AN    #MovElevador.EnPisoAbajo;
      JC    Posicionar_CARGA;


// --- Posicionar en el PUESTO DE TRABAJO
      SET;
      A     #MAQ_Cargada;  // Esta CARGADA
      AN    #FinDesPaletizado;  // Sin ORDEN
      AN    #UT_Datos.SinUT;  // Hay UT
      AN    #UT_Datos.OK_DestinoUT;  // No tiene DESTINO
      A     #UT_Datos.Con_DestinoUT;
      A     #MovElevador.EnPisoAbajo;
      AN    #Robot_Habilitado;
      JC    Posicionar_ARRIBA_SIN_ROBOT;

      SET;
      A     #MAQ_Cargada;  // Esta CARGADA
      AN    #FinDesPaletizado;  // Sin ORDEN
      AN    #UT_Datos.SinUT;  // Hay UT
      AN    #UT_Datos.OK_DestinoUT;  // No tiene DESTINO
      A     #UT_Datos.Con_DestinoUT;
      A     #MovElevador.EnPisoAbajo;
      A     #Robot_Habilitado;
      JC    Posicionar_ARRIBA_CON_ROBOT;


// --- Posicionar para DESCARGAR
      SET;
      A     #MAQ_Cargada;  // Esta CARGADA
      A     #FinDesPaletizado;  // Con ORDEN
      AN    #UT_Datos.SinUT;  // Hay UT
      AN    #MovElevador.EnPisoAbajo;
      JC    Posicionar_DESCARGA;

      SET;
      A     #MAQ_Cargada;  // Esta CARGADA
      AN    #FinDesPaletizado;  // Sin ORDEN
      AN    #UT_Datos.SinUT;  // Hay UT
      A     #UT_Datos.OK_DestinoUT;  // Tiene DESTINO
      A     #UT_Datos.Con_DestinoUT;
      AN    #MovElevador.EnPisoAbajo;
      JC    Posicionar_DESCARGA;

      JU    Final_ControlOrdenes;  // No hay Ordenes



NETWORK
TITLE = ---- Ejecutar Ordenes de Posicionado
/////////////////////////////////////////////////////////////////////////////
/////////////////////////////////////////////////////////////////////////////
/////////////////////////////////////////////////////////////////////////////
/////////////////////////////////////////////////////////////////////////////
// ---  POSICIONAR PARA LA CARGA
Posicionar_CARGA:NOP   0;
      SET;
      S     #Orden;

      L     #ConfigMAQ.PosicionCarga;  // --- Enviar orden de Reposo
      T     #PosicionDOWN;  //     Piso de ABAJO
      T     #PosicionOrden;
      T     #PosicionUltima;

      JU    Final_ControlOrdenes;


/////////////////////////////////////////////////////////////////////////////
/////////////////////////////////////////////////////////////////////////////
/////////////////////////////////////////////////////////////////////////////
/////////////////////////////////////////////////////////////////////////////
// ---  POSICIONAR PARA LA DESCARGA
Posicionar_DESCARGA:NOP   0;
      SET;
      S     #Orden;

      L     #ConfigMAQ.PosicionDesCarga;  // --- Enviar orden de Reposo
      T     #PosicionDOWN;  //     Piso de ABAJO
      T     #PosicionOrden;
      T     #PosicionUltima;

      JU    Final_ControlOrdenes;


/////////////////////////////////////////////////////////////////////////////
/////////////////////////////////////////////////////////////////////////////
/////////////////////////////////////////////////////////////////////////////
/////////////////////////////////////////////////////////////////////////////
// ---  POSICIONAR EN EL PUESTO DE TRABAJO >>> SIN ROBOT
Posicionar_ARRIBA_SIN_ROBOT:NOP   0;
      SET;
      S     #Orden;

      L     #ConfigMAQ.AlturaMax;  // --- Altura Inicial en el Puesto de Trabajo
      L     #UT_Datos.CotaUT;  //     Altura a posicionarse =
      -I;  // = AlturaMaxima - Cota
      L     #UT_Datos.CapaUT;  // + Capa
      +I;
      L     #ConfigMAQ.AlturaPaleta;  // + Altura de Paleta
      +I;
      T     #MovElevador.NuevaPosicion;

//--- Altura Maxima ?
      L     #MovElevador.NuevaPosicion;  // --- Comprueba que no sobrepasa
      L     #ConfigMAQ.AlturaMax;  //     la altura maxima
      <=I;
      JC    MaximoOK_Posicionar_ARRIBA_SIN_ROBOT;

      L     #ConfigMAQ.AlturaMax;  // Lo maximo que se posiciona
      T     #MovElevador.NuevaPosicion;  // para trabajar

MaximoOK_Posicionar_ARRIBA_SIN_ROBOT:NOP   0;
      L     #MovElevador.NuevaPosicion;
      T     #PosicionUP;
      T     #PosicionOrden;
      T     #PosicionUltima;

      JU    Final_ControlOrdenes;
/////////////////////////////////////////////////////////////////////////////
/////////////////////////////////////////////////////////////////////////////
/////////////////////////////////////////////////////////////////////////////
/////////////////////////////////////////////////////////////////////////////
// ---  POSICIONAR EN EL PUESTO DE TRABAJO >>> SIN ROBOT
Posicionar_ARRIBA_CON_ROBOT:NOP   0;
      SET;
      S     #Orden;

      L     #ConfigMAQ.AlturaMax;  // --- Altura Inicial en el Puesto de Trabajo
      L     #UT_Datos.CotaUT;  //     Altura a posicionarse =
      -I;  // = AlturaMaxima - Cota
//      L     #UT_Datos.CapaUT     // + Capa
//      +I
      L     #ConfigMAQ.AlturaPaleta;  // + Altura de Paleta
      +I;
      T     #MovElevador.NuevaPosicion;

//--- Altura Maxima ?
      L     #MovElevador.NuevaPosicion;  // --- Comprueba que no sobrepasa
      L     #ConfigMAQ.AlturaMax;  //     la altura maxima
      <=I;
      JC    MaximoOK_Posicionar_ARRIBA_CON_ROBOT;

      L     #ConfigMAQ.AlturaMax;  // Lo maximo que se posiciona
      T     #MovElevador.NuevaPosicion;  // para trabajar

MaximoOK_Posicionar_ARRIBA_CON_ROBOT:NOP   0;
      L     #MovElevador.NuevaPosicion;
      T     #PosicionUP;
      T     #PosicionOrden;
      T     #PosicionUltima;

      JU    Final_ControlOrdenes;



NETWORK
TITLE = ---- Final
/////////////////////////////////////////////////////////////////////////////
/////////////////////////////////////////////////////////////////////////////
/////////////////////////////////////////////////////////////////////////////
/////////////////////////////////////////////////////////////////////////////
// --- Final del Control de Ordenes
Final_ControlOrdenes:NOP   0;



REGION Network 31: CONTROL DE FRENCUENCIA DE POSICIONADO DEL VATIADOR DEL ELEVADOR
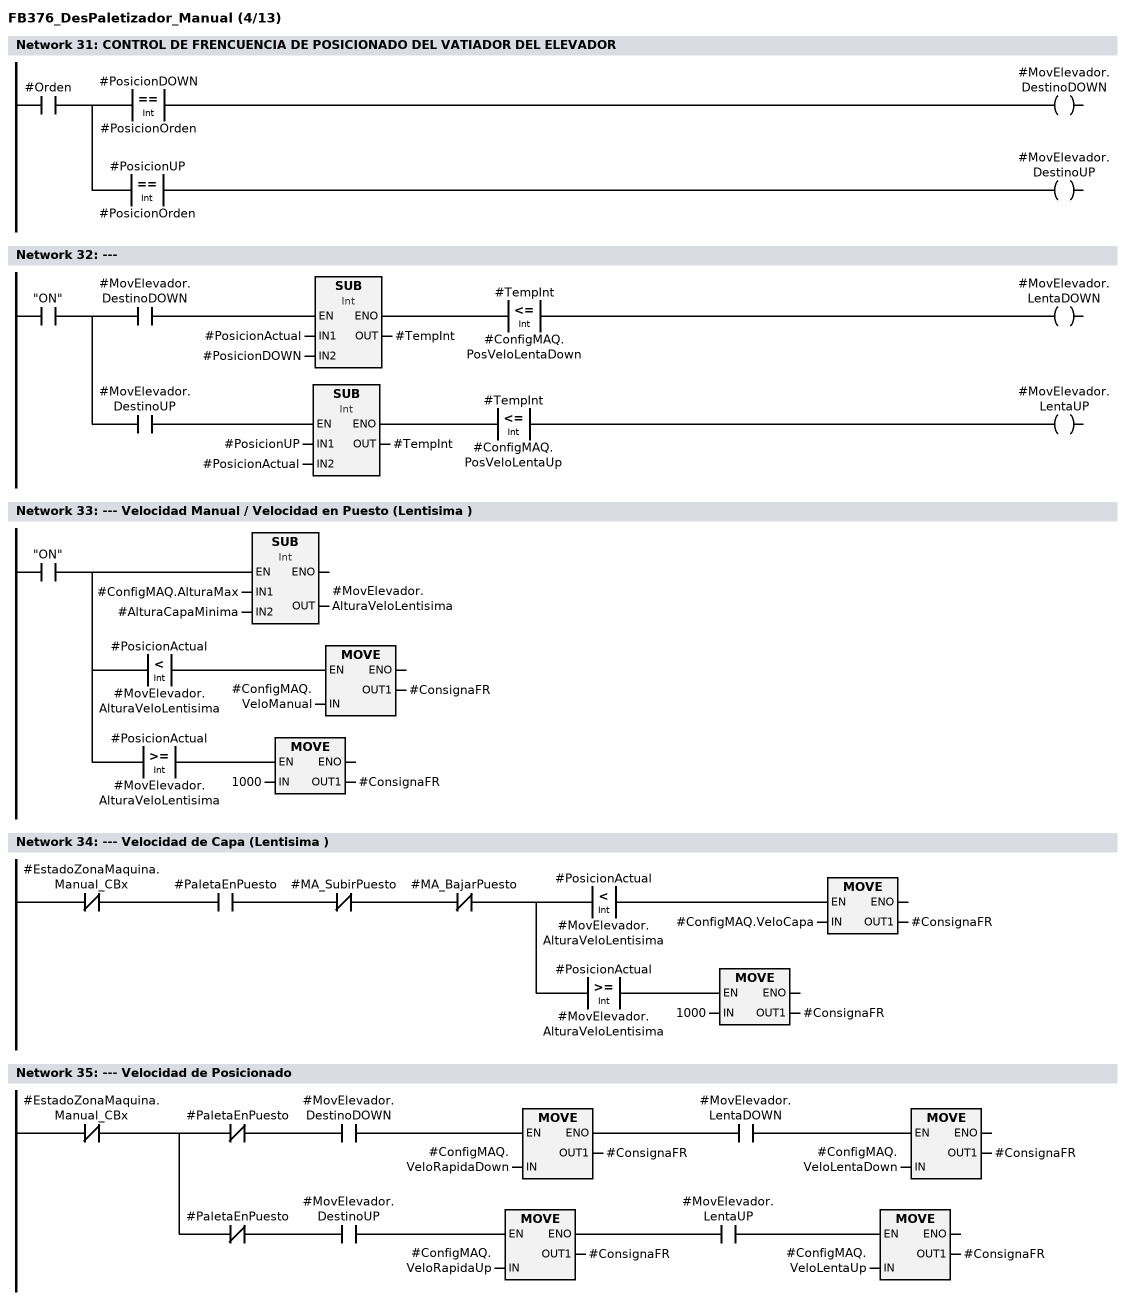
   RUNG wire#powerrail
      Contact( #Orden )
      wire#w1
      { S7_Templates := "SrcType := Int" } EQ_Contact(in1 := #PosicionDOWN, in2 := #PosicionOrden)
      Coil( #MovElevador.DestinoDOWN )
   END_RUNG
   RUNG wire#w1
      { S7_Templates := "SrcType := Int" } EQ_Contact(in1 := #PosicionUP, in2 := #PosicionOrden)
      Coil( #MovElevador.DestinoUP )
   END_RUNG
   // the same network as SCL:
   #MovElevador.DestinoDOWN := #Orden AND (#PosicionDOWN = #PosicionOrden);
   #MovElevador.DestinoUP := #Orden AND (#PosicionUP = #PosicionOrden);
END_REGION

REGION Network 32: ---
   RUNG wire#powerrail
      Contact( "ON" )
      wire#w1
      Contact( #MovElevador.DestinoDOWN )
      { S7_Templates := "SrcType := Int"; S7_GenerateENO := "TRUE" } Sub(in1 := #PosicionActual, in2 := #PosicionDOWN, out => #TempInt)
      { S7_Templates := "SrcType := Int" } LE_Contact(in1 := #TempInt, in2 := #ConfigMAQ.PosVeloLentaDown)
      Coil( #MovElevador.LentaDOWN )
   END_RUNG
   RUNG wire#w1
      Contact( #MovElevador.DestinoUP )
      { S7_Templates := "SrcType := Int"; S7_GenerateENO := "TRUE" } Sub(in1 := #PosicionUP, in2 := #PosicionActual, out => #TempInt)
      { S7_Templates := "SrcType := Int" } LE_Contact(in1 := #TempInt, in2 := #ConfigMAQ.PosVeloLentaUp)
      Coil( #MovElevador.LentaUP )
   END_RUNG
   // the same network as SCL:
   // ENO of a box is taken as its EN; it also drops when the box reports an error
   #_w1 := "ON" AND #MovElevador.DestinoDOWN;
   IF #_w1 THEN #TempInt := #PosicionActual - #PosicionDOWN; END_IF;
   #MovElevador.LentaDOWN := #_w1 AND (#TempInt <= #ConfigMAQ.PosVeloLentaDown);
   #_w2 := "ON" AND #MovElevador.DestinoUP;
   IF #_w2 THEN #TempInt := #PosicionUP - #PosicionActual; END_IF;
   #MovElevador.LentaUP := #_w2 AND (#TempInt <= #ConfigMAQ.PosVeloLentaUp);
END_REGION

REGION Network 33: --- Velocidad Manual / Velocidad en Puesto (Lentisima )
   RUNG wire#powerrail
      Contact( "ON" )
      wire#w1
      { S7_Templates := "SrcType := Int"; S7_GenerateENO := "TRUE" } Sub(in1 := #ConfigMAQ.AlturaMax, in2 := #AlturaCapaMinima, out => #MovElevador.AlturaVeloLentisima)
   END_RUNG
   RUNG wire#w1
      { S7_Templates := "SrcType := Int" } LT_Contact(in1 := #PosicionActual, in2 := #MovElevador.AlturaVeloLentisima)
      { S7_GenerateENO := "TRUE" } Move(in := #ConfigMAQ.VeloManual, out1 => #ConsignaFR)
   END_RUNG
   RUNG wire#w1
      { S7_Templates := "SrcType := Int" } GE_Contact(in1 := #PosicionActual, in2 := #MovElevador.AlturaVeloLentisima)
      { S7_GenerateENO := "TRUE" } Move(in := 1000, out1 => #ConsignaFR)
   END_RUNG
   // the same network as SCL:
   IF "ON" THEN #MovElevador.AlturaVeloLentisima := #ConfigMAQ.AlturaMax - #AlturaCapaMinima; END_IF;
   IF "ON" AND (#PosicionActual < #MovElevador.AlturaVeloLentisima) THEN
       #ConsignaFR := #ConfigMAQ.VeloManual;
   END_IF;
   IF "ON" AND (#PosicionActual >= #MovElevador.AlturaVeloLentisima) THEN #ConsignaFR := 1000; END_IF;
END_REGION

REGION Network 34: --- Velocidad de Capa (Lentisima )
   RUNG wire#powerrail
      I_Contact( #EstadoZonaMaquina.Manual_CBx )
      Contact( #PaletaEnPuesto )
      I_Contact( #MA_SubirPuesto )
      I_Contact( #MA_BajarPuesto )
      wire#w1
      { S7_Templates := "SrcType := Int" } LT_Contact(in1 := #PosicionActual, in2 := #MovElevador.AlturaVeloLentisima)
      { S7_GenerateENO := "TRUE" } Move(in := #ConfigMAQ.VeloCapa, out1 => #ConsignaFR)
   END_RUNG
   RUNG wire#w1
      { S7_Templates := "SrcType := Int" } GE_Contact(in1 := #PosicionActual, in2 := #MovElevador.AlturaVeloLentisima)
      { S7_GenerateENO := "TRUE" } Move(in := 1000, out1 => #ConsignaFR)
   END_RUNG
   // the same network as SCL:
   #_w1 := NOT #EstadoZonaMaquina.Manual_CBx AND #PaletaEnPuesto AND NOT #MA_SubirPuesto AND NOT #MA_BajarPuesto;
   IF #_w1 AND (#PosicionActual < #MovElevador.AlturaVeloLentisima) THEN
       #ConsignaFR := #ConfigMAQ.VeloCapa;
   END_IF;
   IF #_w1 AND (#PosicionActual >= #MovElevador.AlturaVeloLentisima) THEN #ConsignaFR := 1000; END_IF;
END_REGION

REGION Network 35: --- Velocidad de Posicionado
   RUNG wire#powerrail
      I_Contact( #EstadoZonaMaquina.Manual_CBx )
      wire#w1
      I_Contact( #PaletaEnPuesto )
      Contact( #MovElevador.DestinoDOWN )
      { S7_GenerateENO := "TRUE" } Move(in := #ConfigMAQ.VeloRapidaDown, out1 => #ConsignaFR)
      Contact( #MovElevador.LentaDOWN )
      { S7_GenerateENO := "TRUE" } Move(in := #ConfigMAQ.VeloLentaDown, out1 => #ConsignaFR)
   END_RUNG
   RUNG wire#w1
      I_Contact( #PaletaEnPuesto )
      Contact( #MovElevador.DestinoUP )
      { S7_GenerateENO := "TRUE" } Move(in := #ConfigMAQ.VeloRapidaUp, out1 => #ConsignaFR)
      Contact( #MovElevador.LentaUP )
      { S7_GenerateENO := "TRUE" } Move(in := #ConfigMAQ.VeloLentaUp, out1 => #ConsignaFR)
   END_RUNG
   // the same network as SCL:
   // ENO of a box is taken as its EN; it also drops when the box reports an error
   #_w1 := NOT #EstadoZonaMaquina.Manual_CBx;
   #_w2 := #_w1 AND NOT #PaletaEnPuesto AND #MovElevador.DestinoDOWN;
   IF #_w2 THEN #ConsignaFR := #ConfigMAQ.VeloRapidaDown; END_IF;
   IF #_w2 AND #MovElevador.LentaDOWN THEN #ConsignaFR := #ConfigMAQ.VeloLentaDown; END_IF;
   #_w3 := #_w1 AND NOT #PaletaEnPuesto AND #MovElevador.DestinoUP;
   IF #_w3 THEN #ConsignaFR := #ConfigMAQ.VeloRapidaUp; END_IF;
   IF #_w3 AND #MovElevador.LentaUP THEN #ConsignaFR := #ConfigMAQ.VeloLentaUp; END_IF;
END_REGION

REGION Network 36: --- Velocidad de Homing
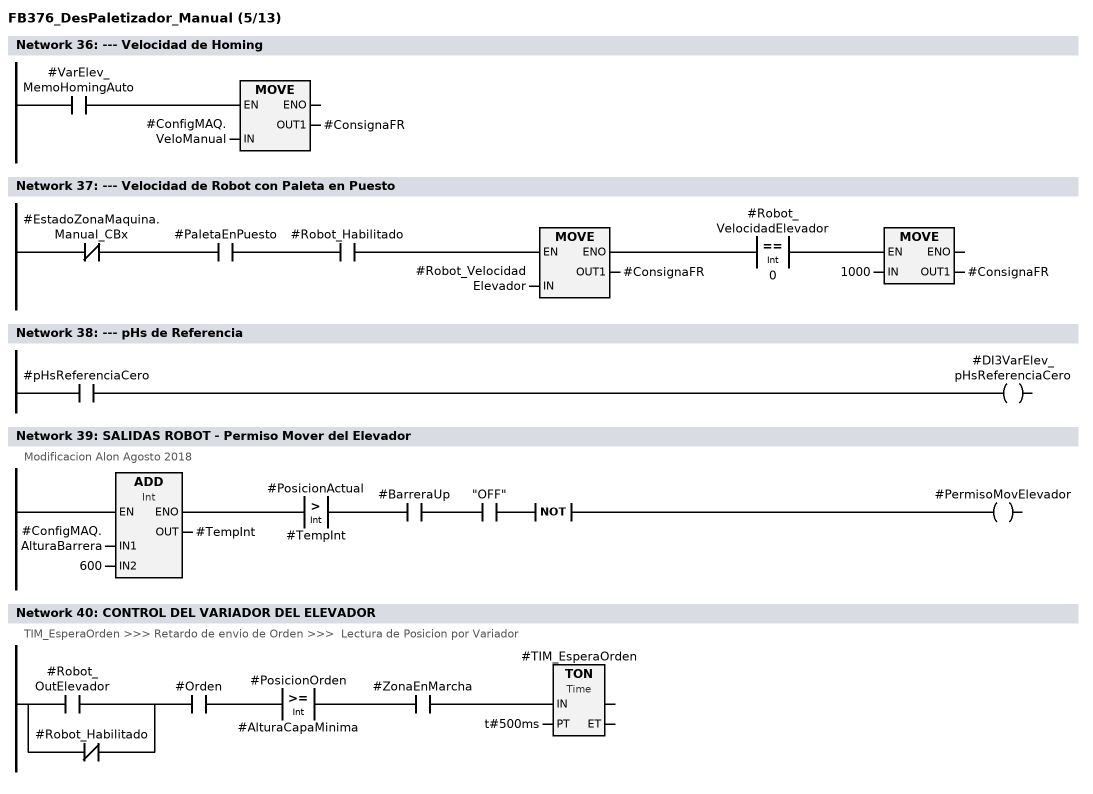
   RUNG wire#powerrail
      Contact( #VarElev_MemoHomingAuto )
      { S7_GenerateENO := "TRUE" } Move(in := #ConfigMAQ.VeloManual, out1 => #ConsignaFR)
   END_RUNG
   // the same network as SCL:
   IF #VarElev_MemoHomingAuto THEN #ConsignaFR := #ConfigMAQ.VeloManual; END_IF;
END_REGION

REGION Network 37: --- Velocidad de Robot con Paleta en Puesto
   RUNG wire#powerrail
      I_Contact( #EstadoZonaMaquina.Manual_CBx )
      Contact( #PaletaEnPuesto )
      Contact( #Robot_Habilitado )
      { S7_GenerateENO := "TRUE" } Move(in := #Robot_VelocidadElevador, out1 => #ConsignaFR)
      { S7_Templates := "SrcType := Int" } EQ_Contact(in1 := #Robot_VelocidadElevador, in2 := 0)
      { S7_GenerateENO := "TRUE" } Move(in := 1000, out1 => #ConsignaFR)
   END_RUNG
   // the same network as SCL:
   // ENO of a box is taken as its EN; it also drops when the box reports an error
   #_w1 := NOT #EstadoZonaMaquina.Manual_CBx AND #PaletaEnPuesto AND #Robot_Habilitado;
   IF #_w1 THEN #ConsignaFR := #Robot_VelocidadElevador; END_IF;
   IF #_w1 AND (#Robot_VelocidadElevador = 0) THEN #ConsignaFR := 1000; END_IF;
END_REGION

REGION Network 38: --- pHs de Referencia
   RUNG wire#powerrail
      Contact( #pHsReferenciaCero )
      Coil( #DI3VarElev_pHsReferenciaCero )
   END_RUNG
   // the same network as SCL:
   #DI3VarElev_pHsReferenciaCero := #pHsReferenciaCero;
END_REGION

REGION Network 39: SALIDAS ROBOT - Permiso Mover del Elevador
   // Modificacion Alon Agosto 2018
   RUNG wire#powerrail
      { S7_Templates := "SrcType := Int"; S7_GenerateENO := "TRUE" } Add(in1 := #ConfigMAQ.AlturaBarrera, in2 := 600, out => #TempInt)
      { S7_Templates := "SrcType := Int" } GT_Contact(in1 := #PosicionActual, in2 := #TempInt)
      Contact( #BarreraUp )
      Contact( "OFF" )
      Not()
      Coil( #PermisoMovElevador )
   END_RUNG
   // the same network as SCL:
   // ENO of a box is taken as its EN; it also drops when the box reports an error
   #TempInt := #ConfigMAQ.AlturaBarrera + 600;
   #PermisoMovElevador := NOT ((#PosicionActual > #TempInt) AND #BarreraUp AND "OFF");
END_REGION

REGION Network 40: CONTROL DEL VARIADOR DEL ELEVADOR
   // TIM_EsperaOrden >>> Retardo de envio de Orden >>>  Lectura de Posicion por Variador
   RUNG wire#powerrail
      Contact( #Robot_OutElevador )
      wire#w1
      Contact( #Orden )
      { S7_Templates := "SrcType := Int" } GE_Contact(in1 := #PosicionOrden, in2 := #AlturaCapaMinima)
      Contact( #ZonaEnMarcha )
      { S7_Templates := "time_type := Time" } #TIM_EsperaOrden.TON(pt := t#500ms, et =>)
   END_RUNG
   RUNG wire#powerrail
      I_Contact( #Robot_Habilitado )
   END_RUNG wire#w1
   // the same network as SCL:
   #TIM_EsperaOrden(IN := (#Robot_OutElevador OR NOT #Robot_Habilitado) AND #Orden AND (#PosicionOrden >= #AlturaCapaMinima) AND #ZonaEnMarcha,   // TON
                    PT := t#500ms);
END_REGION

REGION Network 41: ---- VARIADOR LENZE
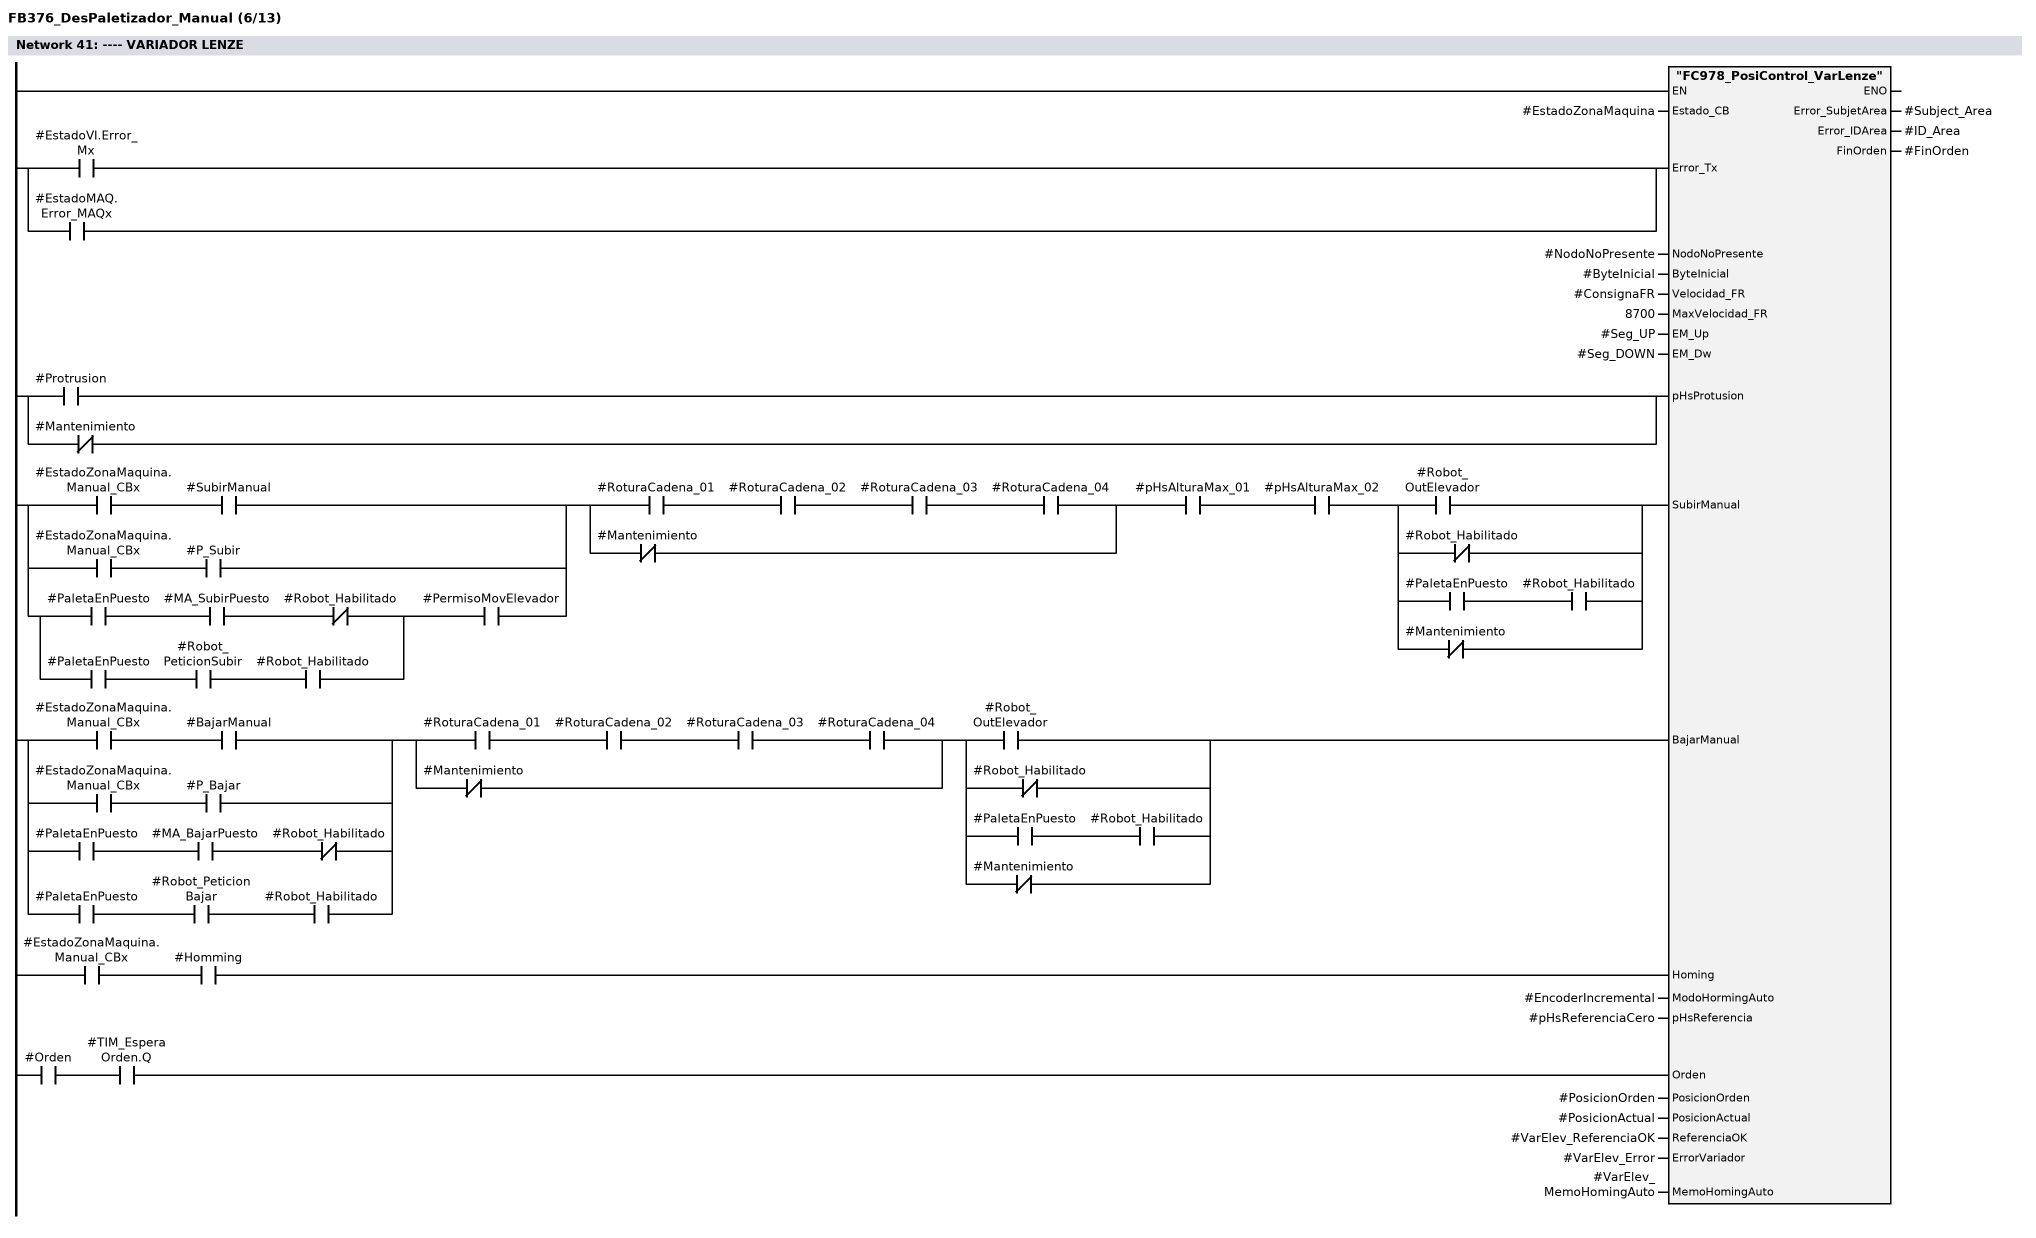
   RUNG wire#powerrail
      "FC978_PosiControl_VarLenze"(Error_Tx := wire#w1, pHsProtusion := wire#w2, SubirManual := wire#w7, BajarManual := wire#w10, Homing := wire#w11, Orden := wire#w12, Estado_CB := #EstadoZonaMaquina, NodoNoPresente := #NodoNoPresente, ByteInicial := #ByteInicial, Velocidad_FR := #ConsignaFR, MaxVelocidad_FR := 8700, EM_Up := #Seg_UP, EM_Dw := #Seg_DOWN, ModoHormingAuto := #EncoderIncremental, pHsReferencia := #pHsReferenciaCero, PosicionOrden := #PosicionOrden, PosicionActual := #PosicionActual, ReferenciaOK := #VarElev_ReferenciaOK, ErrorVariador := #VarElev_Error, MemoHomingAuto := #VarElev_MemoHomingAuto, Error_SubjetArea => #Subject_Area, Error_IDArea => #ID_Area, FinOrden => #FinOrden)
   END_RUNG
   RUNG wire#powerrail
      Contact( #EstadoVI.Error_Mx )
   END_RUNG wire#w1
   RUNG wire#powerrail
      Contact( #EstadoMAQ.Error_MAQx )
   END_RUNG wire#w1
   RUNG wire#powerrail
      Contact( #Protrusion )
   END_RUNG wire#w2
   RUNG wire#powerrail
      I_Contact( #Mantenimiento )
   END_RUNG wire#w2
   RUNG wire#powerrail
      Contact( #EstadoZonaMaquina.Manual_CBx )
      Contact( #SubirManual )
      wire#w3
      Contact( #RoturaCadena_01 )
      Contact( #RoturaCadena_02 )
      Contact( #RoturaCadena_03 )
      Contact( #RoturaCadena_04 )
      wire#w5
      Contact( #pHsAlturaMax_01 )
      Contact( #pHsAlturaMax_02 )
      wire#w6
      Contact( #Robot_OutElevador )
   END_RUNG wire#w7
   RUNG wire#powerrail
      Contact( #EstadoZonaMaquina.Manual_CBx )
      Contact( #P_Subir )
   END_RUNG wire#w3
   RUNG wire#powerrail
      Contact( #PaletaEnPuesto )
      Contact( #MA_SubirPuesto )
      I_Contact( #Robot_Habilitado )
      wire#w4
      Contact( #PermisoMovElevador )
   END_RUNG wire#w3
   RUNG wire#powerrail
      Contact( #PaletaEnPuesto )
      Contact( #Robot_PeticionSubir )
      Contact( #Robot_Habilitado )
   END_RUNG wire#w4
   RUNG wire#w3
      I_Contact( #Mantenimiento )
   END_RUNG wire#w5
   RUNG wire#w6
      I_Contact( #Robot_Habilitado )
   END_RUNG wire#w7
   RUNG wire#w6
      Contact( #PaletaEnPuesto )
      Contact( #Robot_Habilitado )
   END_RUNG wire#w7
   RUNG wire#w6
      I_Contact( #Mantenimiento )
   END_RUNG wire#w7
   RUNG wire#powerrail
      Contact( #EstadoZonaMaquina.Manual_CBx )
      Contact( #BajarManual )
      wire#w8
      Contact( #RoturaCadena_01 )
      Contact( #RoturaCadena_02 )
      Contact( #RoturaCadena_03 )
      Contact( #RoturaCadena_04 )
      wire#w9
      Contact( #Robot_OutElevador )
   END_RUNG wire#w10
   RUNG wire#powerrail
      Contact( #EstadoZonaMaquina.Manual_CBx )
      Contact( #P_Bajar )
   END_RUNG wire#w8
   RUNG wire#powerrail
      Contact( #PaletaEnPuesto )
      Contact( #MA_BajarPuesto )
      I_Contact( #Robot_Habilitado )
   END_RUNG wire#w8
   RUNG wire#powerrail
      Contact( #PaletaEnPuesto )
      Contact( #Robot_PeticionBajar )
      Contact( #Robot_Habilitado )
   END_RUNG wire#w8
   RUNG wire#w8
      I_Contact( #Mantenimiento )
   END_RUNG wire#w9
   RUNG wire#w9
      I_Contact( #Robot_Habilitado )
   END_RUNG wire#w10
   RUNG wire#w9
      Contact( #PaletaEnPuesto )
      Contact( #Robot_Habilitado )
   END_RUNG wire#w10
   RUNG wire#w9
      I_Contact( #Mantenimiento )
   END_RUNG wire#w10
   RUNG wire#powerrail
      Contact( #EstadoZonaMaquina.Manual_CBx )
      Contact( #Homming )
   END_RUNG wire#w11
   RUNG wire#powerrail
      Contact( #Orden )
      Contact( #TIM_EsperaOrden.Q )
   END_RUNG wire#w12
   // the same network as SCL:
   "FC978_PosiControl_VarLenze"(Estado_CB := #EstadoZonaMaquina,
                           Error_Tx := #EstadoVI.Error_Mx OR #EstadoMAQ.Error_MAQx,
                           NodoNoPresente := #NodoNoPresente,
                           ByteInicial := #ByteInicial,
                           Velocidad_FR := #ConsignaFR,
                           MaxVelocidad_FR := 8700,
                           EM_Up := #Seg_UP,
                           EM_Dw := #Seg_DOWN,
                           pHsProtusion := #Protrusion OR NOT #Mantenimiento,
                           SubirManual := ((#EstadoZonaMaquina.Manual_CBx AND #SubirManual) OR (#EstadoZonaMaquina.Manual_CBx AND #P_Subir) OR (((#PaletaEnPuesto AND #MA_SubirPuesto AND NOT #Robot_Habilitado) OR (#PaletaEnPuesto AND #Robot_PeticionSubir AND #Robot_Habilitado)) AND #PermisoMovElevador)) AND ((#RoturaCadena_01 AND #RoturaCadena_02 AND #RoturaCadena_03 AND #RoturaCadena_04) OR NOT #Mantenimiento) AND #pHsAlturaMax_01 AND #pHsAlturaMax_02 AND (#Robot_OutElevador OR NOT #Robot_Habilitado OR (#PaletaEnPuesto AND #Robot_Habilitado) OR NOT #Mantenimiento),
                           BajarManual := ((#EstadoZonaMaquina.Manual_CBx AND #BajarManual) OR (#EstadoZonaMaquina.Manual_CBx AND #P_Bajar) OR (#PaletaEnPuesto AND #MA_BajarPuesto AND NOT #Robot_Habilitado) OR (#PaletaEnPuesto AND #Robot_PeticionBajar AND #Robot_Habilitado)) AND ((#RoturaCadena_01 AND #RoturaCadena_02 AND #RoturaCadena_03 AND #RoturaCadena_04) OR NOT #Mantenimiento) AND (#Robot_OutElevador OR NOT #Robot_Habilitado OR (#PaletaEnPuesto AND #Robot_Habilitado) OR NOT #Mantenimiento),
                           Homing := #EstadoZonaMaquina.Manual_CBx AND #Homming,
                           ModoHormingAuto := #EncoderIncremental,
                           pHsReferencia := #pHsReferenciaCero,
                           Orden := #Orden AND #TIM_EsperaOrden.Q,
                           PosicionOrden := #PosicionOrden,
                           PosicionActual := #PosicionActual,
                           ReferenciaOK := #VarElev_ReferenciaOK,
                           ErrorVariador := #VarElev_Error,
                           MemoHomingAuto := #VarElev_MemoHomingAuto,
                           Error_SubjetArea => #Subject_Area,
                           Error_IDArea => #ID_Area,
                           FinOrden => #FinOrden);
END_REGION

REGION Network 42: EVENTO DE PALETIZADO >>> INICIO DE DESPALETIZADO
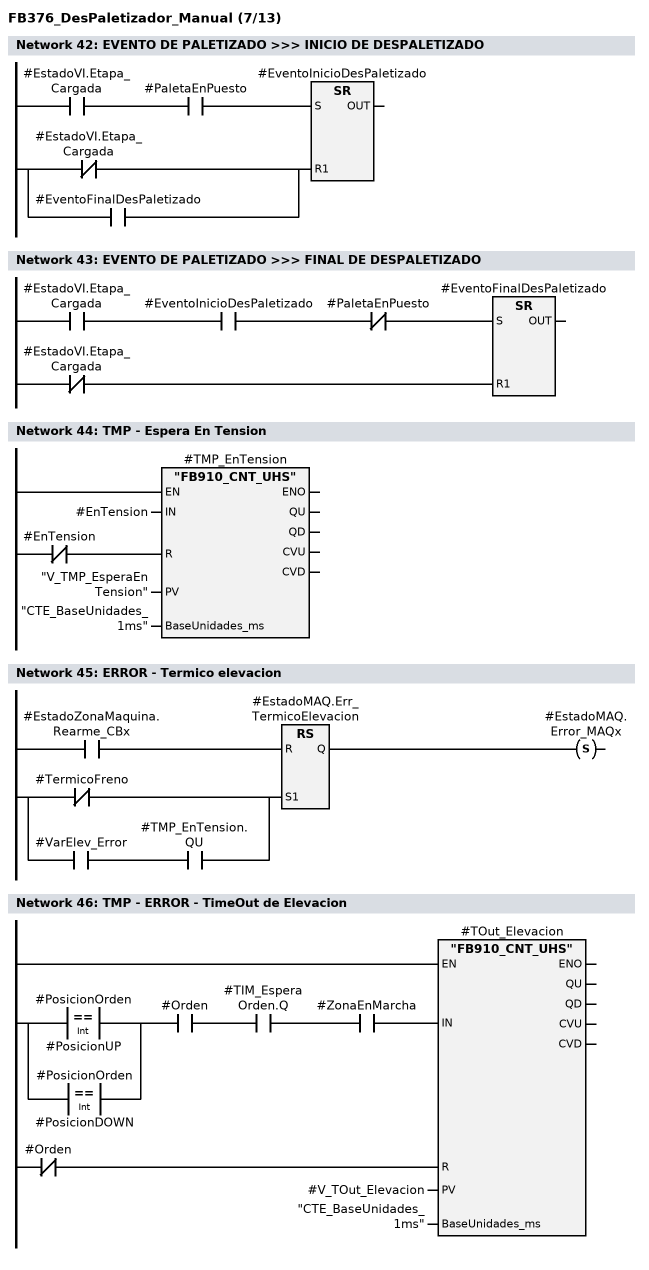
   RUNG wire#powerrail
      Contact( #EstadoVI.Etapa_Cargada )
      Contact( #PaletaEnPuesto )
      S_SR(operand := #EventoInicioDesPaletizado, r1 := wire#w1)
   END_RUNG
   RUNG wire#powerrail
      I_Contact( #EstadoVI.Etapa_Cargada )
   END_RUNG wire#w1
   RUNG wire#powerrail
      Contact( #EventoFinalDesPaletizado )
   END_RUNG wire#w1
   // the same network as SCL:
   IF #EstadoVI.Etapa_Cargada AND #PaletaEnPuesto THEN
       #EventoInicioDesPaletizado := TRUE;   // SR flip-flop
   END_IF;
   IF NOT #EstadoVI.Etapa_Cargada OR #EventoFinalDesPaletizado THEN
       #EventoInicioDesPaletizado := FALSE;
   END_IF;
END_REGION

REGION Network 43: EVENTO DE PALETIZADO >>> FINAL DE DESPALETIZADO
   RUNG wire#powerrail
      Contact( #EstadoVI.Etapa_Cargada )
      Contact( #EventoInicioDesPaletizado )
      I_Contact( #PaletaEnPuesto )
      S_SR(operand := #EventoFinalDesPaletizado, r1 := wire#w1)
   END_RUNG
   RUNG wire#powerrail
      I_Contact( #EstadoVI.Etapa_Cargada )
   END_RUNG wire#w1
   // the same network as SCL:
   IF #EstadoVI.Etapa_Cargada AND #EventoInicioDesPaletizado AND NOT #PaletaEnPuesto THEN
       #EventoFinalDesPaletizado := TRUE;   // SR flip-flop
   END_IF;
   IF NOT #EstadoVI.Etapa_Cargada THEN #EventoFinalDesPaletizado := FALSE; END_IF;
END_REGION

REGION Network 44: TMP - Espera En Tension
   RUNG wire#powerrail
      #TMP_EnTension(R := wire#w1, IN := #EnTension, PV := "V_TMP_EsperaEnTension", BaseUnidades_ms := "CTE_BaseUnidades_1ms", QU =>, QD =>, CVU =>, CVD =>)
   END_RUNG
   RUNG wire#powerrail
      I_Contact( #EnTension )
   END_RUNG wire#w1
   // the same network as SCL:
   #TMP_EnTension(IN := #EnTension,   // "FB910_CNT_UHS"
                  R := NOT #EnTension,
                  PV := "V_TMP_EsperaEnTension",
                  BaseUnidades_ms := "CTE_BaseUnidades_1ms");
END_REGION

REGION Network 45: ERROR - Termico elevacion
   RUNG wire#powerrail
      Contact( #EstadoZonaMaquina.Rearme_CBx )
      S_RS(operand := #EstadoMAQ.Err_TermicoElevacion, s1 := wire#w1)
      S_Coil( #EstadoMAQ.Error_MAQx )
   END_RUNG
   RUNG wire#powerrail
      I_Contact( #TermicoFreno )
   END_RUNG wire#w1
   RUNG wire#powerrail
      Contact( #VarElev_Error )
      Contact( #TMP_EnTension.QU )
   END_RUNG wire#w1
   // the same network as SCL:
   IF #EstadoZonaMaquina.Rearme_CBx THEN
       #EstadoMAQ.Err_TermicoElevacion := FALSE;   // RS flip-flop
   END_IF;
   IF NOT #TermicoFreno OR (#VarElev_Error AND #TMP_EnTension.QU) THEN
       #EstadoMAQ.Err_TermicoElevacion := TRUE;
   END_IF;
   IF #EstadoMAQ.Err_TermicoElevacion THEN #EstadoMAQ.Error_MAQx := TRUE; END_IF;
END_REGION

REGION Network 46: TMP - ERROR - TimeOut de Elevacion
   RUNG wire#powerrail
      #TOut_Elevacion(IN := wire#w2, R := wire#w3, PV := #V_TOut_Elevacion, BaseUnidades_ms := "CTE_BaseUnidades_1ms", QU =>, QD =>, CVU =>, CVD =>)
   END_RUNG
   RUNG wire#powerrail
      { S7_Templates := "SrcType := Int" } EQ_Contact(in1 := #PosicionOrden, in2 := #PosicionUP)
      wire#w1
      Contact( #Orden )
      Contact( #TIM_EsperaOrden.Q )
      Contact( #ZonaEnMarcha )
   END_RUNG wire#w2
   RUNG wire#powerrail
      { S7_Templates := "SrcType := Int" } EQ_Contact(in1 := #PosicionOrden, in2 := #PosicionDOWN)
   END_RUNG wire#w1
   RUNG wire#powerrail
      I_Contact( #Orden )
   END_RUNG wire#w3
   // the same network as SCL:
   #TOut_Elevacion(IN := ((#PosicionOrden = #PosicionUP) OR (#PosicionOrden = #PosicionDOWN)) AND #Orden AND #TIM_EsperaOrden.Q AND #ZonaEnMarcha,   // "FB910_CNT_UHS"
                   R := NOT #Orden,
                   PV := #V_TOut_Elevacion,
                   BaseUnidades_ms := "CTE_BaseUnidades_1ms");
END_REGION

REGION Network 47: ERROR - TimeOut de Elevacion
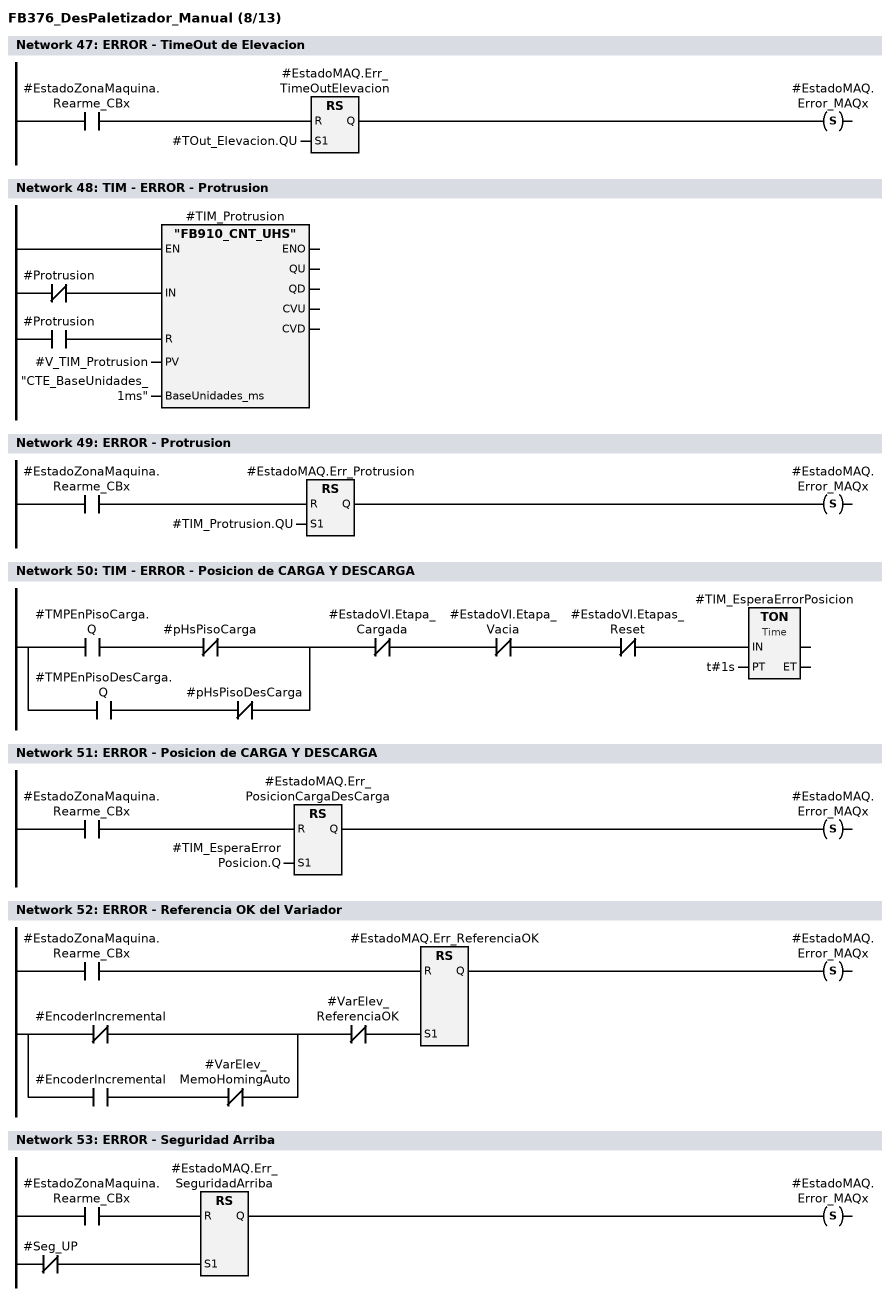
   RUNG wire#powerrail
      Contact( #EstadoZonaMaquina.Rearme_CBx )
      S_RS(operand := #EstadoMAQ.Err_TimeOutElevacion, s1 := #TOut_Elevacion.QU)
      S_Coil( #EstadoMAQ.Error_MAQx )
   END_RUNG
   // the same network as SCL:
   IF #EstadoZonaMaquina.Rearme_CBx THEN
       #EstadoMAQ.Err_TimeOutElevacion := FALSE;   // RS flip-flop
   END_IF;
   IF #TOut_Elevacion.QU THEN #EstadoMAQ.Err_TimeOutElevacion := TRUE; END_IF;
   IF #EstadoMAQ.Err_TimeOutElevacion THEN #EstadoMAQ.Error_MAQx := TRUE; END_IF;
END_REGION

REGION Network 48: TIM - ERROR - Protrusion
   RUNG wire#powerrail
      #TIM_Protrusion(IN := wire#w1, R := wire#w2, PV := #V_TIM_Protrusion, BaseUnidades_ms := "CTE_BaseUnidades_1ms", QU =>, QD =>, CVU =>, CVD =>)
   END_RUNG
   RUNG wire#powerrail
      I_Contact( #Protrusion )
   END_RUNG wire#w1
   RUNG wire#powerrail
      Contact( #Protrusion )
   END_RUNG wire#w2
   // the same network as SCL:
   #TIM_Protrusion(IN := NOT #Protrusion,   // "FB910_CNT_UHS"
                   R := #Protrusion,
                   PV := #V_TIM_Protrusion,
                   BaseUnidades_ms := "CTE_BaseUnidades_1ms");
END_REGION

REGION Network 49: ERROR - Protrusion
   RUNG wire#powerrail
      Contact( #EstadoZonaMaquina.Rearme_CBx )
      S_RS(operand := #EstadoMAQ.Err_Protrusion, s1 := #TIM_Protrusion.QU)
      S_Coil( #EstadoMAQ.Error_MAQx )
   END_RUNG
   // the same network as SCL:
   IF #EstadoZonaMaquina.Rearme_CBx THEN
       #EstadoMAQ.Err_Protrusion := FALSE;   // RS flip-flop
   END_IF;
   IF #TIM_Protrusion.QU THEN #EstadoMAQ.Err_Protrusion := TRUE; END_IF;
   IF #EstadoMAQ.Err_Protrusion THEN #EstadoMAQ.Error_MAQx := TRUE; END_IF;
END_REGION

REGION Network 50: TIM - ERROR - Posicion de CARGA Y DESCARGA
   RUNG wire#powerrail
      Contact( #TMPEnPisoCarga.Q )
      I_Contact( #pHsPisoCarga )
      wire#w1
      I_Contact( #EstadoVI.Etapa_Cargada )
      I_Contact( #EstadoVI.Etapa_Vacia )
      I_Contact( #EstadoVI.Etapas_Reset )
      { S7_Templates := "time_type := Time" } #TIM_EsperaErrorPosicion.TON(pt := t#1s, et =>)
   END_RUNG
   RUNG wire#powerrail
      Contact( #TMPEnPisoDesCarga.Q )
      I_Contact( #pHsPisoDesCarga )
   END_RUNG wire#w1
   // the same network as SCL:
   #TIM_EsperaErrorPosicion(IN := ((#TMPEnPisoCarga.Q AND NOT #pHsPisoCarga) OR (#TMPEnPisoDesCarga.Q AND NOT #pHsPisoDesCarga)) AND NOT #EstadoVI.Etapa_Cargada AND NOT #EstadoVI.Etapa_Vacia AND NOT #EstadoVI.Etapas_Reset,   // TON
                           PT := t#1s);
END_REGION

REGION Network 51: ERROR - Posicion de CARGA Y DESCARGA
   RUNG wire#powerrail
      Contact( #EstadoZonaMaquina.Rearme_CBx )
      S_RS(operand := #EstadoMAQ.Err_PosicionCargaDesCarga, s1 := #TIM_EsperaErrorPosicion.Q)
      S_Coil( #EstadoMAQ.Error_MAQx )
   END_RUNG
   // the same network as SCL:
   IF #EstadoZonaMaquina.Rearme_CBx THEN
       #EstadoMAQ.Err_PosicionCargaDesCarga := FALSE;   // RS flip-flop
   END_IF;
   IF #TIM_EsperaErrorPosicion.Q THEN #EstadoMAQ.Err_PosicionCargaDesCarga := TRUE; END_IF;
   IF #EstadoMAQ.Err_PosicionCargaDesCarga THEN #EstadoMAQ.Error_MAQx := TRUE; END_IF;
END_REGION

REGION Network 52: ERROR - Referencia OK del Variador
   RUNG wire#powerrail
      Contact( #EstadoZonaMaquina.Rearme_CBx )
      S_RS(operand := #EstadoMAQ.Err_ReferenciaOK, s1 := wire#w2)
      S_Coil( #EstadoMAQ.Error_MAQx )
   END_RUNG
   RUNG wire#powerrail
      I_Contact( #EncoderIncremental )
      wire#w1
      I_Contact( #VarElev_ReferenciaOK )
   END_RUNG wire#w2
   RUNG wire#powerrail
      Contact( #EncoderIncremental )
      I_Contact( #VarElev_MemoHomingAuto )
   END_RUNG wire#w1
   // the same network as SCL:
   IF #EstadoZonaMaquina.Rearme_CBx THEN
       #EstadoMAQ.Err_ReferenciaOK := FALSE;   // RS flip-flop
   END_IF;
   IF (NOT #EncoderIncremental OR (#EncoderIncremental AND NOT #VarElev_MemoHomingAuto)) AND NOT #VarElev_ReferenciaOK THEN
       #EstadoMAQ.Err_ReferenciaOK := TRUE;
   END_IF;
   IF #EstadoMAQ.Err_ReferenciaOK THEN #EstadoMAQ.Error_MAQx := TRUE; END_IF;
END_REGION

REGION Network 53: ERROR - Seguridad Arriba
   RUNG wire#powerrail
      Contact( #EstadoZonaMaquina.Rearme_CBx )
      S_RS(operand := #EstadoMAQ.Err_SeguridadArriba, s1 := wire#w1)
      S_Coil( #EstadoMAQ.Error_MAQx )
   END_RUNG
   RUNG wire#powerrail
      I_Contact( #Seg_UP )
   END_RUNG wire#w1
   // the same network as SCL:
   IF #EstadoZonaMaquina.Rearme_CBx THEN
       #EstadoMAQ.Err_SeguridadArriba := FALSE;   // RS flip-flop
   END_IF;
   IF NOT #Seg_UP THEN #EstadoMAQ.Err_SeguridadArriba := TRUE; END_IF;
   IF #EstadoMAQ.Err_SeguridadArriba THEN #EstadoMAQ.Error_MAQx := TRUE; END_IF;
END_REGION

REGION Network 54: ERROR - Seguridad Abajo
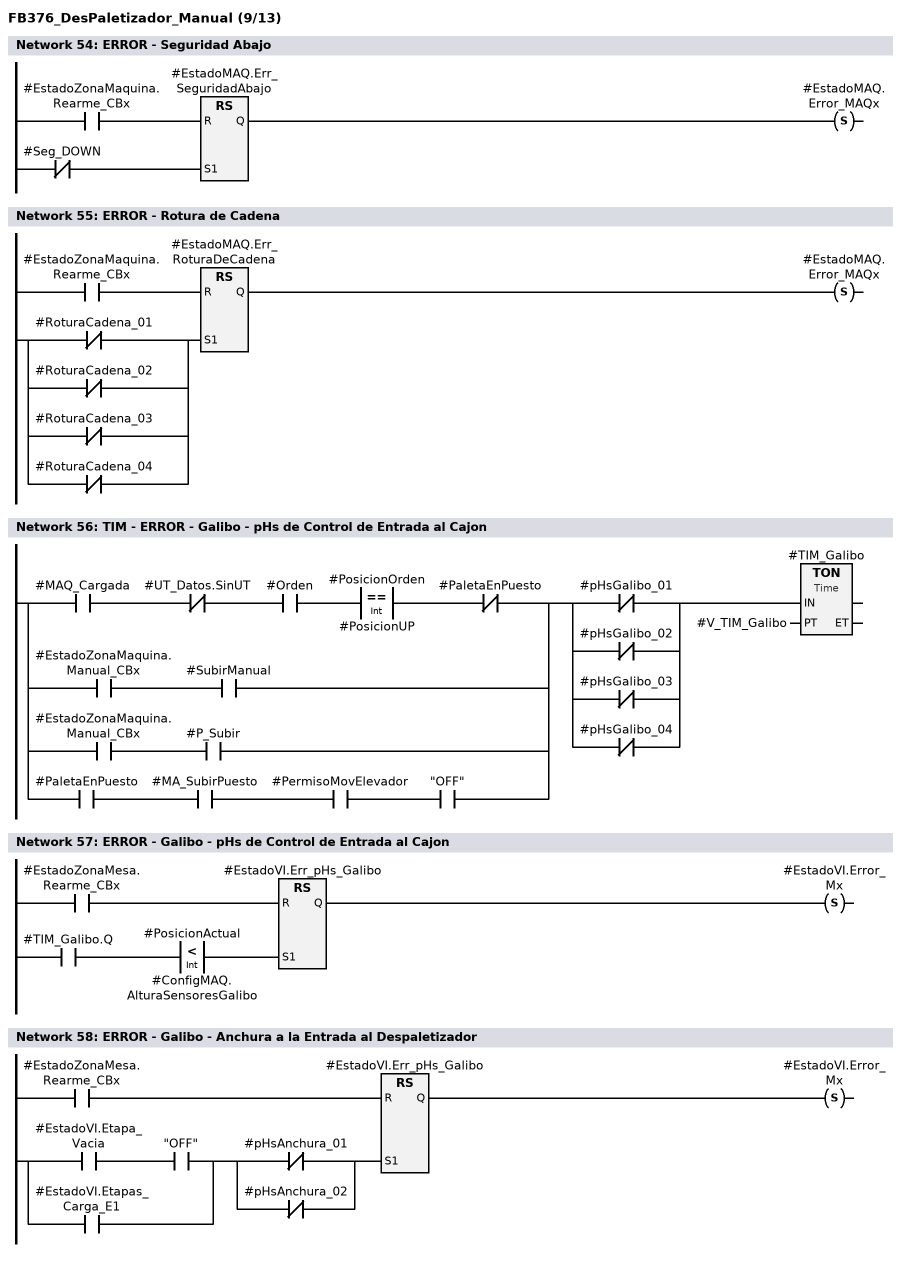
   RUNG wire#powerrail
      Contact( #EstadoZonaMaquina.Rearme_CBx )
      S_RS(operand := #EstadoMAQ.Err_SeguridadAbajo, s1 := wire#w1)
      S_Coil( #EstadoMAQ.Error_MAQx )
   END_RUNG
   RUNG wire#powerrail
      I_Contact( #Seg_DOWN )
   END_RUNG wire#w1
   // the same network as SCL:
   IF #EstadoZonaMaquina.Rearme_CBx THEN
       #EstadoMAQ.Err_SeguridadAbajo := FALSE;   // RS flip-flop
   END_IF;
   IF NOT #Seg_DOWN THEN #EstadoMAQ.Err_SeguridadAbajo := TRUE; END_IF;
   IF #EstadoMAQ.Err_SeguridadAbajo THEN #EstadoMAQ.Error_MAQx := TRUE; END_IF;
END_REGION

REGION Network 55: ERROR - Rotura de Cadena
   RUNG wire#powerrail
      Contact( #EstadoZonaMaquina.Rearme_CBx )
      S_RS(operand := #EstadoMAQ.Err_RoturaDeCadena, s1 := wire#w1)
      S_Coil( #EstadoMAQ.Error_MAQx )
   END_RUNG
   RUNG wire#powerrail
      I_Contact( #RoturaCadena_01 )
   END_RUNG wire#w1
   RUNG wire#powerrail
      I_Contact( #RoturaCadena_02 )
   END_RUNG wire#w1
   RUNG wire#powerrail
      I_Contact( #RoturaCadena_03 )
   END_RUNG wire#w1
   RUNG wire#powerrail
      I_Contact( #RoturaCadena_04 )
   END_RUNG wire#w1
   // the same network as SCL:
   IF #EstadoZonaMaquina.Rearme_CBx THEN
       #EstadoMAQ.Err_RoturaDeCadena := FALSE;   // RS flip-flop
   END_IF;
   IF NOT #RoturaCadena_01 OR NOT #RoturaCadena_02 OR NOT #RoturaCadena_03 OR NOT #RoturaCadena_04 THEN
       #EstadoMAQ.Err_RoturaDeCadena := TRUE;
   END_IF;
   IF #EstadoMAQ.Err_RoturaDeCadena THEN #EstadoMAQ.Error_MAQx := TRUE; END_IF;
END_REGION

REGION Network 56: TIM - ERROR - Galibo - pHs de Control de Entrada al Cajon
   RUNG wire#powerrail
      Contact( #MAQ_Cargada )
      I_Contact( #UT_Datos.SinUT )
      Contact( #Orden )
      { S7_Templates := "SrcType := Int" } EQ_Contact(in1 := #PosicionOrden, in2 := #PosicionUP)
      I_Contact( #PaletaEnPuesto )
      wire#w1
      I_Contact( #pHsGalibo_01 )
      wire#w2
      { S7_Templates := "time_type := Time" } #TIM_Galibo.TON(pt := #V_TIM_Galibo, et =>)
   END_RUNG
   RUNG wire#powerrail
      Contact( #EstadoZonaMaquina.Manual_CBx )
      Contact( #SubirManual )
   END_RUNG wire#w1
   RUNG wire#powerrail
      Contact( #EstadoZonaMaquina.Manual_CBx )
      Contact( #P_Subir )
   END_RUNG wire#w1
   RUNG wire#powerrail
      Contact( #PaletaEnPuesto )
      Contact( #MA_SubirPuesto )
      Contact( #PermisoMovElevador )
      Contact( "OFF" )
   END_RUNG wire#w1
   RUNG wire#w1
      I_Contact( #pHsGalibo_02 )
   END_RUNG wire#w2
   RUNG wire#w1
      I_Contact( #pHsGalibo_03 )
   END_RUNG wire#w2
   RUNG wire#w1
      I_Contact( #pHsGalibo_04 )
   END_RUNG wire#w2
   // the same network as SCL:
   #TIM_Galibo(IN := ((#MAQ_Cargada AND NOT #UT_Datos.SinUT AND #Orden AND (#PosicionOrden = #PosicionUP) AND NOT #PaletaEnPuesto) OR (#EstadoZonaMaquina.Manual_CBx AND #SubirManual) OR (#EstadoZonaMaquina.Manual_CBx AND #P_Subir) OR (#PaletaEnPuesto AND #MA_SubirPuesto AND #PermisoMovElevador AND "OFF")) AND (NOT #pHsGalibo_01 OR NOT #pHsGalibo_02 OR NOT #pHsGalibo_03 OR NOT #pHsGalibo_04),   // TON
               PT := #V_TIM_Galibo);
END_REGION

REGION Network 57: ERROR - Galibo - pHs de Control de Entrada al Cajon
   RUNG wire#powerrail
      Contact( #EstadoZonaMesa.Rearme_CBx )
      S_RS(operand := #EstadoVI.Err_pHs_Galibo, s1 := wire#w1)
      S_Coil( #EstadoVI.Error_Mx )
   END_RUNG
   RUNG wire#powerrail
      Contact( #TIM_Galibo.Q )
      { S7_Templates := "SrcType := Int" } LT_Contact(in1 := #PosicionActual, in2 := #ConfigMAQ.AlturaSensoresGalibo)
   END_RUNG wire#w1
   // the same network as SCL:
   IF #EstadoZonaMesa.Rearme_CBx THEN
       #EstadoVI.Err_pHs_Galibo := FALSE;   // RS flip-flop
   END_IF;
   IF #TIM_Galibo.Q AND (#PosicionActual < #ConfigMAQ.AlturaSensoresGalibo) THEN
       #EstadoVI.Err_pHs_Galibo := TRUE;
   END_IF;
   IF #EstadoVI.Err_pHs_Galibo THEN #EstadoVI.Error_Mx := TRUE; END_IF;
END_REGION

REGION Network 58: ERROR - Galibo - Anchura a la Entrada al Despaletizador
   RUNG wire#powerrail
      Contact( #EstadoZonaMesa.Rearme_CBx )
      S_RS(operand := #EstadoVI.Err_pHs_Galibo, s1 := wire#w2)
      S_Coil( #EstadoVI.Error_Mx )
   END_RUNG
   RUNG wire#powerrail
      Contact( #EstadoVI.Etapa_Vacia )
      Contact( "OFF" )
      wire#w1
      I_Contact( #pHsAnchura_01 )
   END_RUNG wire#w2
   RUNG wire#powerrail
      Contact( #EstadoVI.Etapas_Carga_E1 )
   END_RUNG wire#w1
   RUNG wire#w1
      I_Contact( #pHsAnchura_02 )
   END_RUNG wire#w2
   // the same network as SCL:
   IF #EstadoZonaMesa.Rearme_CBx THEN
       #EstadoVI.Err_pHs_Galibo := FALSE;   // RS flip-flop
   END_IF;
   IF ((#EstadoVI.Etapa_Vacia AND "OFF") OR #EstadoVI.Etapas_Carga_E1) AND (NOT #pHsAnchura_01 OR NOT #pHsAnchura_02) THEN
       #EstadoVI.Err_pHs_Galibo := TRUE;
   END_IF;
   IF #EstadoVI.Err_pHs_Galibo THEN #EstadoVI.Error_Mx := TRUE; END_IF;
END_REGION

REGION Network 59: ERROR - Galibo - Altura al Movimiento Vertical
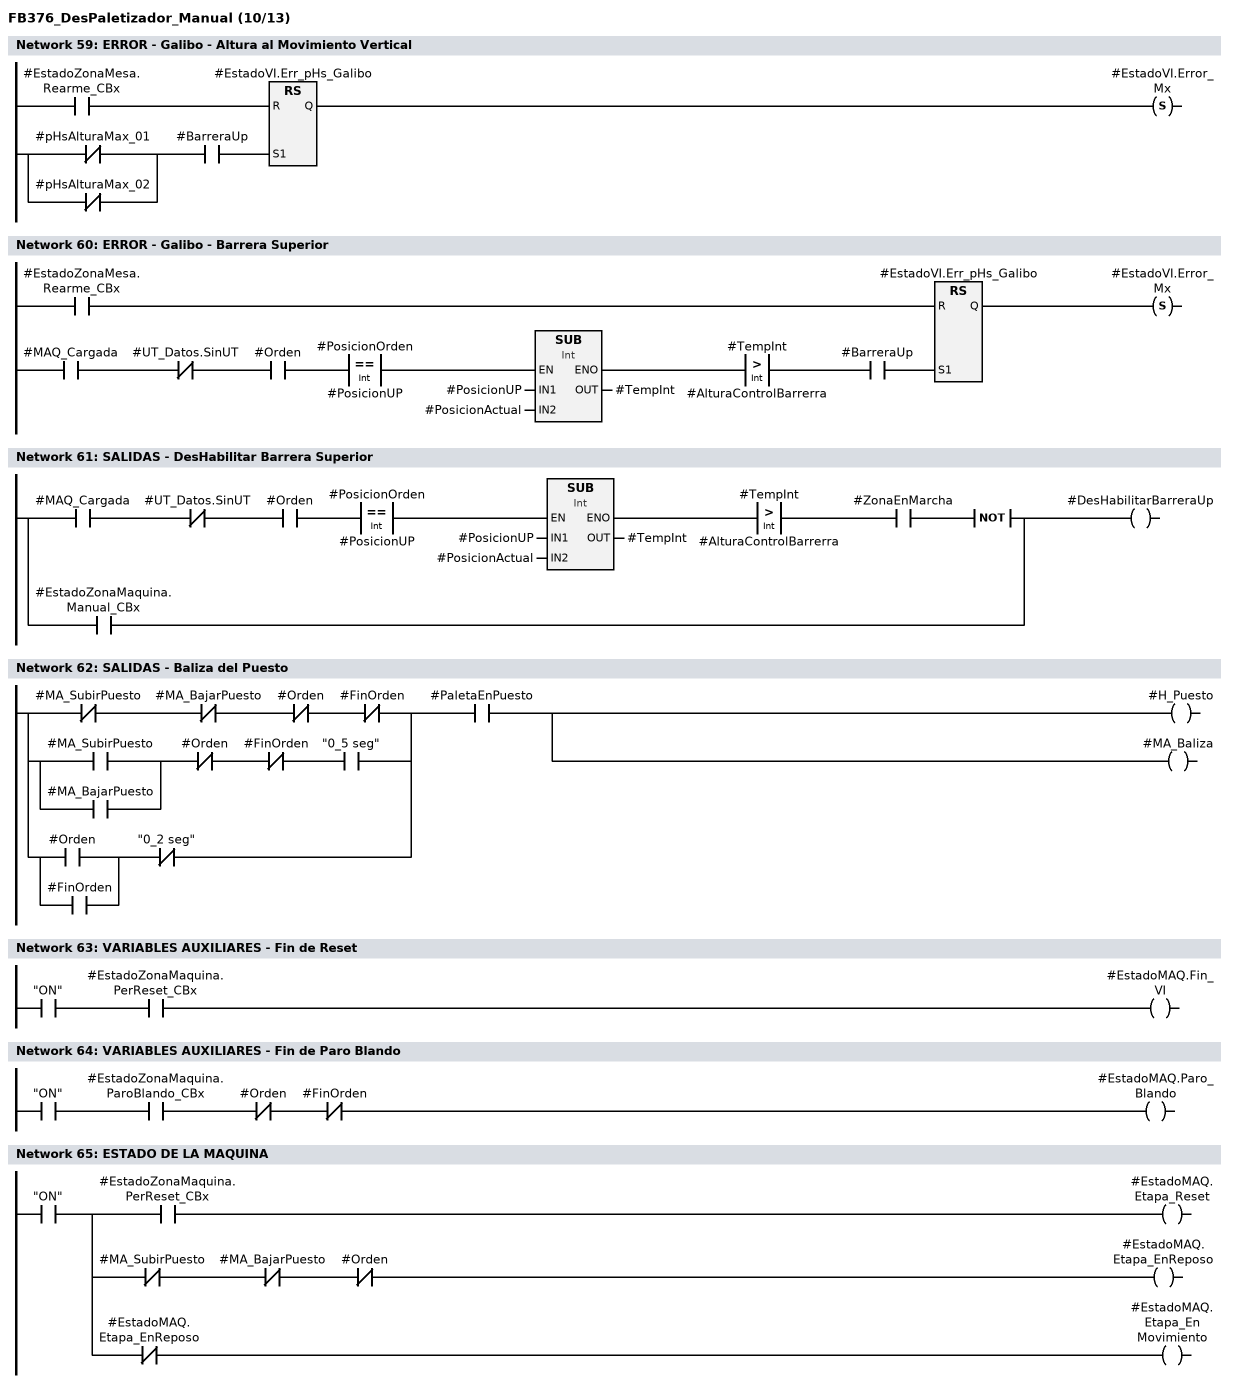
   RUNG wire#powerrail
      Contact( #EstadoZonaMesa.Rearme_CBx )
      S_RS(operand := #EstadoVI.Err_pHs_Galibo, s1 := wire#w2)
      S_Coil( #EstadoVI.Error_Mx )
   END_RUNG
   RUNG wire#powerrail
      I_Contact( #pHsAlturaMax_01 )
      wire#w1
      Contact( #BarreraUp )
   END_RUNG wire#w2
   RUNG wire#powerrail
      I_Contact( #pHsAlturaMax_02 )
   END_RUNG wire#w1
   // the same network as SCL:
   IF #EstadoZonaMesa.Rearme_CBx THEN
       #EstadoVI.Err_pHs_Galibo := FALSE;   // RS flip-flop
   END_IF;
   IF (NOT #pHsAlturaMax_01 OR NOT #pHsAlturaMax_02) AND #BarreraUp THEN
       #EstadoVI.Err_pHs_Galibo := TRUE;
   END_IF;
   IF #EstadoVI.Err_pHs_Galibo THEN #EstadoVI.Error_Mx := TRUE; END_IF;
END_REGION

REGION Network 60: ERROR - Galibo - Barrera Superior
   RUNG wire#powerrail
      Contact( #EstadoZonaMesa.Rearme_CBx )
      S_RS(operand := #EstadoVI.Err_pHs_Galibo, s1 := wire#w1)
      S_Coil( #EstadoVI.Error_Mx )
   END_RUNG
   RUNG wire#powerrail
      Contact( #MAQ_Cargada )
      I_Contact( #UT_Datos.SinUT )
      Contact( #Orden )
      { S7_Templates := "SrcType := Int" } EQ_Contact(in1 := #PosicionOrden, in2 := #PosicionUP)
      { S7_Templates := "SrcType := Int"; S7_GenerateENO := "TRUE" } Sub(in1 := #PosicionUP, in2 := #PosicionActual, out => #TempInt)
      { S7_Templates := "SrcType := Int" } GT_Contact(in1 := #TempInt, in2 := #AlturaControlBarrerra)
      Contact( #BarreraUp )
   END_RUNG wire#w1
   // the same network as SCL:
   // ENO of a box is taken as its EN; it also drops when the box reports an error
   #_w1 := #MAQ_Cargada AND NOT #UT_Datos.SinUT AND #Orden AND (#PosicionOrden = #PosicionUP);
   IF #_w1 THEN #TempInt := #PosicionUP - #PosicionActual; END_IF;
   IF #EstadoZonaMesa.Rearme_CBx THEN
       #EstadoVI.Err_pHs_Galibo := FALSE;   // RS flip-flop
   END_IF;
   IF #_w1 AND (#TempInt > #AlturaControlBarrerra) AND #BarreraUp THEN
       #EstadoVI.Err_pHs_Galibo := TRUE;
   END_IF;
   IF #EstadoVI.Err_pHs_Galibo THEN #EstadoVI.Error_Mx := TRUE; END_IF;
END_REGION

REGION Network 61: SALIDAS - DesHabilitar Barrera Superior
   RUNG wire#powerrail
      Contact( #MAQ_Cargada )
      I_Contact( #UT_Datos.SinUT )
      Contact( #Orden )
      { S7_Templates := "SrcType := Int" } EQ_Contact(in1 := #PosicionOrden, in2 := #PosicionUP)
      { S7_Templates := "SrcType := Int"; S7_GenerateENO := "TRUE" } Sub(in1 := #PosicionUP, in2 := #PosicionActual, out => #TempInt)
      { S7_Templates := "SrcType := Int" } GT_Contact(in1 := #TempInt, in2 := #AlturaControlBarrerra)
      Contact( #ZonaEnMarcha )
      Not()
      wire#w1
      Coil( #DesHabilitarBarreraUp )
   END_RUNG
   RUNG wire#powerrail
      Contact( #EstadoZonaMaquina.Manual_CBx )
   END_RUNG wire#w1
   // the same network as SCL:
   // ENO of a box is taken as its EN; it also drops when the box reports an error
   #_w1 := #MAQ_Cargada AND NOT #UT_Datos.SinUT AND #Orden AND (#PosicionOrden = #PosicionUP);
   IF #_w1 THEN #TempInt := #PosicionUP - #PosicionActual; END_IF;
   #DesHabilitarBarreraUp := NOT (#_w1 AND (#TempInt > #AlturaControlBarrerra) AND #ZonaEnMarcha) OR #EstadoZonaMaquina.Manual_CBx;
END_REGION

REGION Network 62: SALIDAS - Baliza del Puesto
   RUNG wire#powerrail
      I_Contact( #MA_SubirPuesto )
      I_Contact( #MA_BajarPuesto )
      I_Contact( #Orden )
      I_Contact( #FinOrden )
      wire#w1
      Contact( #PaletaEnPuesto )
      wire#w4
      Coil( #H_Puesto )
   END_RUNG
   RUNG wire#powerrail
      Contact( #MA_SubirPuesto )
      wire#w2
      I_Contact( #Orden )
      I_Contact( #FinOrden )
      Contact( "0_5 seg" )
   END_RUNG wire#w1
   RUNG wire#powerrail
      Contact( #MA_BajarPuesto )
   END_RUNG wire#w2
   RUNG wire#powerrail
      Contact( #Orden )
      wire#w3
      I_Contact( "0_2 seg" )
   END_RUNG wire#w1
   RUNG wire#powerrail
      Contact( #FinOrden )
   END_RUNG wire#w3
   RUNG wire#w4
      Coil( #MA_Baliza )
   END_RUNG
   // the same network as SCL:
   #H_Puesto := ((NOT #MA_SubirPuesto AND NOT #MA_BajarPuesto AND NOT #Orden AND NOT #FinOrden) OR ((#MA_SubirPuesto OR #MA_BajarPuesto) AND NOT #Orden AND NOT #FinOrden AND "0_5 seg") OR ((#Orden OR #FinOrden) AND NOT "0_2 seg")) AND #PaletaEnPuesto;
   #MA_Baliza := #H_Puesto;
END_REGION

REGION Network 63: VARIABLES AUXILIARES - Fin de Reset
   RUNG wire#powerrail
      Contact( "ON" )
      Contact( #EstadoZonaMaquina.PerReset_CBx )
      Coil( #EstadoMAQ.Fin_VI )
   END_RUNG
   // the same network as SCL:
   #EstadoMAQ.Fin_VI := "ON" AND #EstadoZonaMaquina.PerReset_CBx;
END_REGION

REGION Network 64: VARIABLES AUXILIARES - Fin de Paro Blando
   RUNG wire#powerrail
      Contact( "ON" )
      Contact( #EstadoZonaMaquina.ParoBlando_CBx )
      I_Contact( #Orden )
      I_Contact( #FinOrden )
      Coil( #EstadoMAQ.Paro_Blando )
   END_RUNG
   // the same network as SCL:
   #EstadoMAQ.Paro_Blando := "ON" AND #EstadoZonaMaquina.ParoBlando_CBx AND NOT #Orden AND NOT #FinOrden;
END_REGION

REGION Network 65: ESTADO DE LA MAQUINA
   RUNG wire#powerrail
      Contact( "ON" )
      wire#w1
      Contact( #EstadoZonaMaquina.PerReset_CBx )
      Coil( #EstadoMAQ.Etapa_Reset )
   END_RUNG
   RUNG wire#w1
      I_Contact( #MA_SubirPuesto )
      I_Contact( #MA_BajarPuesto )
      I_Contact( #Orden )
      Coil( #EstadoMAQ.Etapa_EnReposo )
   END_RUNG
   RUNG wire#w1
      I_Contact( #EstadoMAQ.Etapa_EnReposo )
      Coil( #EstadoMAQ.Etapa_EnMovimiento )
   END_RUNG
   // the same network as SCL:
   #EstadoMAQ.Etapa_Reset := "ON" AND #EstadoZonaMaquina.PerReset_CBx;
   #EstadoMAQ.Etapa_EnReposo := "ON" AND NOT #MA_SubirPuesto AND NOT #MA_BajarPuesto AND NOT #Orden;
   #EstadoMAQ.Etapa_EnMovimiento := "ON" AND NOT #EstadoMAQ.Etapa_EnReposo;
END_REGION

REGION Network 66: ---
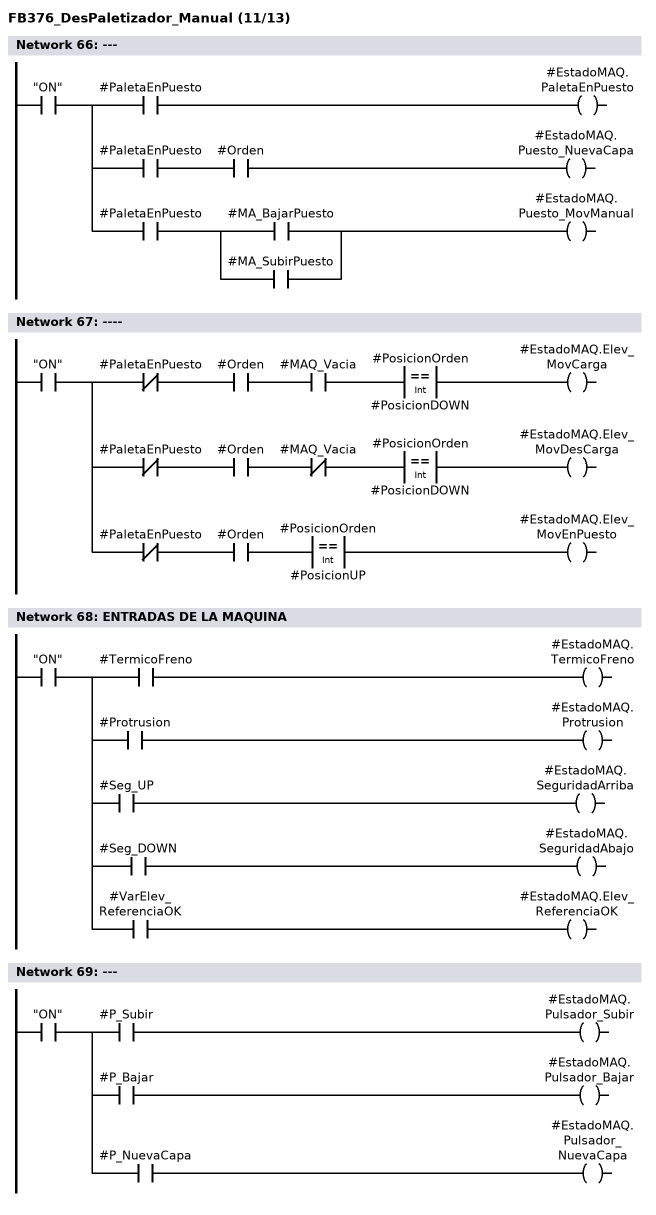
   RUNG wire#powerrail
      Contact( "ON" )
      wire#w1
      Contact( #PaletaEnPuesto )
      Coil( #EstadoMAQ.PaletaEnPuesto )
   END_RUNG
   RUNG wire#w1
      Contact( #PaletaEnPuesto )
      Contact( #Orden )
      Coil( #EstadoMAQ.Puesto_NuevaCapa )
   END_RUNG
   RUNG wire#w1
      Contact( #PaletaEnPuesto )
      wire#w2
      Contact( #MA_BajarPuesto )
      wire#w3
      Coil( #EstadoMAQ.Puesto_MovManual )
   END_RUNG
   RUNG wire#w2
      Contact( #MA_SubirPuesto )
   END_RUNG wire#w3
   // the same network as SCL:
   #EstadoMAQ.PaletaEnPuesto := "ON" AND #PaletaEnPuesto;
   #EstadoMAQ.Puesto_NuevaCapa := "ON" AND #PaletaEnPuesto AND #Orden;
   #EstadoMAQ.Puesto_MovManual := "ON" AND #PaletaEnPuesto AND (#MA_BajarPuesto OR #MA_SubirPuesto);
END_REGION

REGION Network 67: ----
   RUNG wire#powerrail
      Contact( "ON" )
      wire#w1
      I_Contact( #PaletaEnPuesto )
      Contact( #Orden )
      Contact( #MAQ_Vacia )
      { S7_Templates := "SrcType := Int" } EQ_Contact(in1 := #PosicionOrden, in2 := #PosicionDOWN)
      Coil( #EstadoMAQ.Elev_MovCarga )
   END_RUNG
   RUNG wire#w1
      I_Contact( #PaletaEnPuesto )
      Contact( #Orden )
      I_Contact( #MAQ_Vacia )
      { S7_Templates := "SrcType := Int" } EQ_Contact(in1 := #PosicionOrden, in2 := #PosicionDOWN)
      Coil( #EstadoMAQ.Elev_MovDesCarga )
   END_RUNG
   RUNG wire#w1
      I_Contact( #PaletaEnPuesto )
      Contact( #Orden )
      { S7_Templates := "SrcType := Int" } EQ_Contact(in1 := #PosicionOrden, in2 := #PosicionUP)
      Coil( #EstadoMAQ.Elev_MovEnPuesto )
   END_RUNG
   // the same network as SCL:
   #EstadoMAQ.Elev_MovCarga := "ON" AND NOT #PaletaEnPuesto AND #Orden AND #MAQ_Vacia AND (#PosicionOrden = #PosicionDOWN);
   #EstadoMAQ.Elev_MovDesCarga := "ON" AND NOT #PaletaEnPuesto AND #Orden AND NOT #MAQ_Vacia AND (#PosicionOrden = #PosicionDOWN);
   #EstadoMAQ.Elev_MovEnPuesto := "ON" AND NOT #PaletaEnPuesto AND #Orden AND (#PosicionOrden = #PosicionUP);
END_REGION

REGION Network 68: ENTRADAS DE LA MAQUINA
   RUNG wire#powerrail
      Contact( "ON" )
      wire#w1
      Contact( #TermicoFreno )
      Coil( #EstadoMAQ.TermicoFreno )
   END_RUNG
   RUNG wire#w1
      Contact( #Protrusion )
      Coil( #EstadoMAQ.Protrusion )
   END_RUNG
   RUNG wire#w1
      Contact( #Seg_UP )
      Coil( #EstadoMAQ.SeguridadArriba )
   END_RUNG
   RUNG wire#w1
      Contact( #Seg_DOWN )
      Coil( #EstadoMAQ.SeguridadAbajo )
   END_RUNG
   RUNG wire#w1
      Contact( #VarElev_ReferenciaOK )
      Coil( #EstadoMAQ.Elev_ReferenciaOK )
   END_RUNG
   // the same network as SCL:
   #EstadoMAQ.TermicoFreno := "ON" AND #TermicoFreno;
   #EstadoMAQ.Protrusion := "ON" AND #Protrusion;
   #EstadoMAQ.SeguridadArriba := "ON" AND #Seg_UP;
   #EstadoMAQ.SeguridadAbajo := "ON" AND #Seg_DOWN;
   #EstadoMAQ.Elev_ReferenciaOK := "ON" AND #VarElev_ReferenciaOK;
END_REGION

REGION Network 69: ---
   RUNG wire#powerrail
      Contact( "ON" )
      wire#w1
      Contact( #P_Subir )
      Coil( #EstadoMAQ.Pulsador_Subir )
   END_RUNG
   RUNG wire#w1
      Contact( #P_Bajar )
      Coil( #EstadoMAQ.Pulsador_Bajar )
   END_RUNG
   RUNG wire#w1
      Contact( #P_NuevaCapa )
      Coil( #EstadoMAQ.Pulsador_NuevaCapa )
   END_RUNG
   // the same network as SCL:
   #EstadoMAQ.Pulsador_Subir := "ON" AND #P_Subir;
   #EstadoMAQ.Pulsador_Bajar := "ON" AND #P_Bajar;
   #EstadoMAQ.Pulsador_NuevaCapa := "ON" AND #P_NuevaCapa;
END_REGION

REGION Network 70: ---
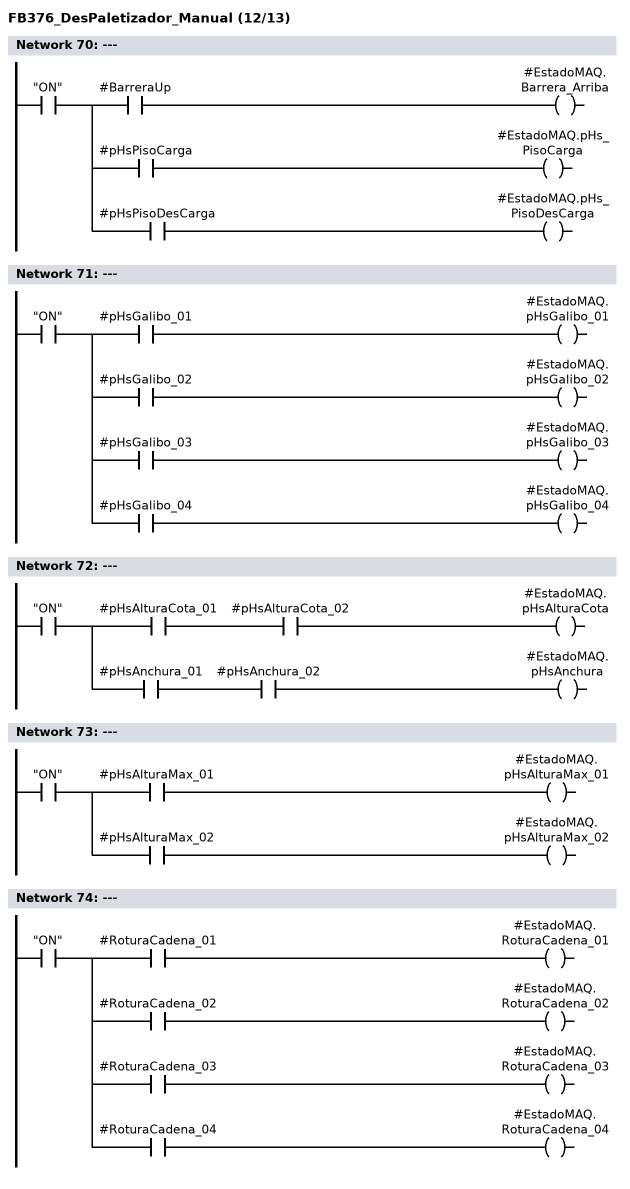
   RUNG wire#powerrail
      Contact( "ON" )
      wire#w1
      Contact( #BarreraUp )
      Coil( #EstadoMAQ.Barrera_Arriba )
   END_RUNG
   RUNG wire#w1
      Contact( #pHsPisoCarga )
      Coil( #EstadoMAQ.pHs_PisoCarga )
   END_RUNG
   RUNG wire#w1
      Contact( #pHsPisoDesCarga )
      Coil( #EstadoMAQ.pHs_PisoDesCarga )
   END_RUNG
   // the same network as SCL:
   #EstadoMAQ.Barrera_Arriba := "ON" AND #BarreraUp;
   #EstadoMAQ.pHs_PisoCarga := "ON" AND #pHsPisoCarga;
   #EstadoMAQ.pHs_PisoDesCarga := "ON" AND #pHsPisoDesCarga;
END_REGION

REGION Network 71: ---
   RUNG wire#powerrail
      Contact( "ON" )
      wire#w1
      Contact( #pHsGalibo_01 )
      Coil( #EstadoMAQ.pHsGalibo_01 )
   END_RUNG
   RUNG wire#w1
      Contact( #pHsGalibo_02 )
      Coil( #EstadoMAQ.pHsGalibo_02 )
   END_RUNG
   RUNG wire#w1
      Contact( #pHsGalibo_03 )
      Coil( #EstadoMAQ.pHsGalibo_03 )
   END_RUNG
   RUNG wire#w1
      Contact( #pHsGalibo_04 )
      Coil( #EstadoMAQ.pHsGalibo_04 )
   END_RUNG
   // the same network as SCL:
   #EstadoMAQ.pHsGalibo_01 := "ON" AND #pHsGalibo_01;
   #EstadoMAQ.pHsGalibo_02 := "ON" AND #pHsGalibo_02;
   #EstadoMAQ.pHsGalibo_03 := "ON" AND #pHsGalibo_03;
   #EstadoMAQ.pHsGalibo_04 := "ON" AND #pHsGalibo_04;
END_REGION

REGION Network 72: ---
   RUNG wire#powerrail
      Contact( "ON" )
      wire#w1
      Contact( #pHsAlturaCota_01 )
      Contact( #pHsAlturaCota_02 )
      Coil( #EstadoMAQ.pHsAlturaCota )
   END_RUNG
   RUNG wire#w1
      Contact( #pHsAnchura_01 )
      Contact( #pHsAnchura_02 )
      Coil( #EstadoMAQ.pHsAnchura )
   END_RUNG
   // the same network as SCL:
   #EstadoMAQ.pHsAlturaCota := "ON" AND #pHsAlturaCota_01 AND #pHsAlturaCota_02;
   #EstadoMAQ.pHsAnchura := "ON" AND #pHsAnchura_01 AND #pHsAnchura_02;
END_REGION

REGION Network 73: ---
   RUNG wire#powerrail
      Contact( "ON" )
      wire#w1
      Contact( #pHsAlturaMax_01 )
      Coil( #EstadoMAQ.pHsAlturaMax_01 )
   END_RUNG
   RUNG wire#w1
      Contact( #pHsAlturaMax_02 )
      Coil( #EstadoMAQ.pHsAlturaMax_02 )
   END_RUNG
   // the same network as SCL:
   #EstadoMAQ.pHsAlturaMax_01 := "ON" AND #pHsAlturaMax_01;
   #EstadoMAQ.pHsAlturaMax_02 := "ON" AND #pHsAlturaMax_02;
END_REGION

REGION Network 74: ---
   RUNG wire#powerrail
      Contact( "ON" )
      wire#w1
      Contact( #RoturaCadena_01 )
      Coil( #EstadoMAQ.RoturaCadena_01 )
   END_RUNG
   RUNG wire#w1
      Contact( #RoturaCadena_02 )
      Coil( #EstadoMAQ.RoturaCadena_02 )
   END_RUNG
   RUNG wire#w1
      Contact( #RoturaCadena_03 )
      Coil( #EstadoMAQ.RoturaCadena_03 )
   END_RUNG
   RUNG wire#w1
      Contact( #RoturaCadena_04 )
      Coil( #EstadoMAQ.RoturaCadena_04 )
   END_RUNG
   // the same network as SCL:
   #EstadoMAQ.RoturaCadena_01 := "ON" AND #RoturaCadena_01;
   #EstadoMAQ.RoturaCadena_02 := "ON" AND #RoturaCadena_02;
   #EstadoMAQ.RoturaCadena_03 := "ON" AND #RoturaCadena_03;
   #EstadoMAQ.RoturaCadena_04 := "ON" AND #RoturaCadena_04;
END_REGION

REGION Network 75: SALIDAS DE LA MAQUINA
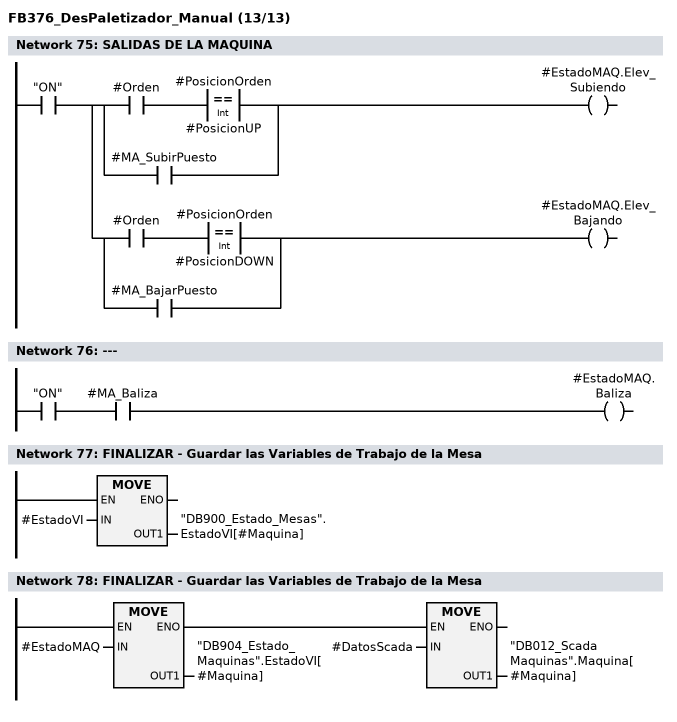
   RUNG wire#powerrail
      Contact( "ON" )
      wire#w1
      Contact( #Orden )
      { S7_Templates := "SrcType := Int" } EQ_Contact(in1 := #PosicionOrden, in2 := #PosicionUP)
      wire#w2
      Coil( #EstadoMAQ.Elev_Subiendo )
   END_RUNG
   RUNG wire#w1
      Contact( #MA_SubirPuesto )
   END_RUNG wire#w2
   RUNG wire#w1
      Contact( #Orden )
      { S7_Templates := "SrcType := Int" } EQ_Contact(in1 := #PosicionOrden, in2 := #PosicionDOWN)
      wire#w3
      Coil( #EstadoMAQ.Elev_Bajando )
   END_RUNG
   RUNG wire#w1
      Contact( #MA_BajarPuesto )
   END_RUNG wire#w3
   // the same network as SCL:
   #EstadoMAQ.Elev_Subiendo := "ON" AND ((#Orden AND (#PosicionOrden = #PosicionUP)) OR #MA_SubirPuesto);
   #EstadoMAQ.Elev_Bajando := "ON" AND ((#Orden AND (#PosicionOrden = #PosicionDOWN)) OR #MA_BajarPuesto);
END_REGION

REGION Network 76: ---
   RUNG wire#powerrail
      Contact( "ON" )
      Contact( #MA_Baliza )
      Coil( #EstadoMAQ.Baliza )
   END_RUNG
   // the same network as SCL:
   #EstadoMAQ.Baliza := "ON" AND #MA_Baliza;
END_REGION

REGION Network 77: FINALIZAR - Guardar las Variables de Trabajo de la Mesa
   RUNG wire#powerrail
      Move(in := #EstadoVI, out1 => "DB900_Estado_Mesas".EstadoVI[#Maquina])
   END_RUNG
   // the same network as SCL:
   "DB900_Estado_Mesas".EstadoVI[#Maquina] := #EstadoVI;
END_REGION

REGION Network 78: FINALIZAR - Guardar las Variables de Trabajo de la Mesa
   RUNG wire#powerrail
      Move(in := #EstadoMAQ, out1 => "DB904_Estado_Maquinas".EstadoVI[#Maquina])
      Move(in := #DatosScada, out1 => "DB012_ScadaMaquinas".Maquina[#Maquina])
   END_RUNG
   // the same network as SCL:
   "DB904_Estado_Maquinas".EstadoVI[#Maquina] := #EstadoMAQ;
   "DB012_ScadaMaquinas".Maquina[#Maquina] := #DatosScada;
END_REGION
END_FUNCTION_BLOCK
